	//arm state machine
	g_stateMachineArm1 : INT;
	g_stateMachineArm2 : INT;
	
	// index(0 to 4) of slave arm which is tele-linked to master arm
	g_teleSlaveArm1Idx : INT;
	g_teleSlaveArm2Idx : INT;
	
	//slave check enable  : true start , false end
	g_slaveCheckEnbale : BOOL;

	//0: init status 1: checking 2:check succeed 3: check failed
	g_slaveCheckStatus : UINT;

	//arm switch 
	g_armSwitchEnable : UINT:=0;

	//master hearbeat  : 1s frequency
	g_heartBeat : INT;

	//screen Lock Enable : true Lock  ,  false  unlock
	g_screenLockEnable : BOOL;
END_VAR

// ---- GVLs/GVL_MathDefine.TcGVL
VAR_GLOBAL CONSTANT
	g_smallNum :LREAL := 1E-8;
	g_smallAng :LREAL := 0.0001*PI/180;
	g_largeNum: LREAL :=1E16;
	g_deg2Rad :LREAL := pi/180.0;
	g_rad2Deg :LREAL := 180.0/pi;
	g_2pi :LREAL := 2*PI;
	
	g_eye3d :Mat3d:=[1, 0, 0,
					 0, 1, 0,
					 0, 0, 1];
	g_eye4d :Mat4d:=[1, 0, 0, 0,
					 0, 1, 0, 0,
					 0, 0, 1, 0,
					 0, 0, 0, 1];
	g_zeroMat3d :Mat3d:=[9(0)];
	
	g_zeroMat6d :Mat6d:=[36(0)];
	g_zeroMat7d :Mat7d:=[49(0)];
	g_eye7d :Mat7d:=[1, 0, 0, 0, 0, 0, 0, 
					 0, 1, 0, 0, 0, 0, 0, 
					 0, 0, 1, 0, 0, 0, 0, 
					 0, 0, 0, 1, 0, 0, 0,
					 0, 0, 0, 0, 1, 0, 0,
					 0, 0, 0, 0, 0, 1, 0,
					 0, 0, 0, 0, 0, 0, 1];
	
	g_zeroVec3d :Vec3d:= [3(0)];
	g_onesVec3d: Vec3d:=[3(1)];
	
	g_zeroVec6d: Vec6d:=[6(0)];
	g_onesVec6d: Vec6d:=[6(1)];
	
	g_zeroVec4d: Vec4d:=[4(0)];
	g_onesVec4d: Vec4d:=[4(1.0)];
	g_zeroVec4i: Vec4i:=[4(0)];
	g_onesVec4i: Vec4i:=[4(1)];
	
	g_zeroVec7d: Vec7d:=[7(0)];
	g_onesVec7d: Vec7d:=[7(1.0)];
	g_zeroVec7i: Vec7i:=[7(0)];
	g_onesVec7i: Vec7i:=[7(1)];
	
	g_allPosMode:Vec7i:=[7(DriverOPMode_Pos)];
	g_allTrqMode:Vec7i:=[7(DriverOPMode_Trq)];
	g_allPosTrqMode:Vec7i:=[7(DriverOPMode_PosTrq)];
	
	
END_VAR

// ---- GVLs/GVL_SafetyParameters.TcGVL
{attribute 'global_init_slot' := '49991'}
//TODO: safety check parameters need to be reviewd
VAR_GLOBAL CONSTANT
	
	// safety error counts threshold to trigger fault
	g_faultTriggerCounts :INT :=2;
	
	// arm joint safety error
	g_armMaxJntEncErr :vec7d:=[7(40*g_deg2Rad)];
	g_armMaxJntFollowErr :vec7d:=[7(20*g_deg2Rad)];
	
	// joint limit buffer(outside of joint limit)
	g_armJntPosLimitBuffer :vec7d:=[3(10.0*g_deg2Rad), 4(45.0*g_deg2Rad)];

	//max joint encoder current  saltation
	g_maxJntCurSalta : vec7di:=[7(60000)];
	
	// self check timeout time limit
	g_selfCheckTimeLimit : LREAL:= 15.0;
	
	//arm joint link encoder maximum and minimum values
	g_maxLinkEnc : DINT:=16777215;
	g_minLinkEnc : DINT:=0;
	
	//drive error word
	g_driveErrWord : UDINT:=32;
	
	// master arm cartesion control safety error 
	g_maxCartPosErr :LREAL := 0.005;
	g_maxCartOriErr :LREAL := 5.0*g_deg2Rad;
	

	// master joint safety error
	g_maxJntCtrlErr :LREAL := 15.0*g_deg2Rad;
	g_maxJntEncErr :LREAL := 30.0*g_deg2Rad;
	
	g_minJntPos: ARRAY[1..2,1..7] OF LREAL:=[-60*g_deg2Rad,	-45*g_deg2Rad-pi/2,		-45*g_deg2Rad, 	0, 	-135*g_deg2Rad+pi,		-45*g_deg2Rad-pi/2,		-g_largeNum,
											 -60*g_deg2Rad,	-45*g_deg2Rad-pi/2,		-45*g_deg2Rad,	0,		-135*g_deg2Rad+pi,		-45*g_deg2Rad+pi/2,	-g_largeNum];
	g_maxJntPos: ARRAY[1..2,1..7] OF LREAL:=[60*g_deg2Rad,	60*g_deg2Rad-pi/2,		60*g_deg2Rad,		2*pi,			135*g_deg2Rad+pi,		45*g_deg2Rad-pi/2,		g_largeNum,
								             60*g_deg2Rad,	60*g_deg2Rad-pi/2,		60*g_deg2Rad,		2*pi,			135*g_deg2Rad+pi,		45*g_deg2Rad+pi/2,		g_largeNum];

	
	// cart joint safety error
	g_cartMaxJntCtrlErr :Vec4d := [0.005, 5*g_deg2Rad,0.005, 0.005];
	g_cartMaxJntEncErr :Vec4d :=  [0.005, 5*g_deg2Rad,0.005, 0.005];

	// cart joint limit buffer(outside of joint limit)
	g_cartJntPosLimitBuffer :Vec4d :=[0.05, 10*g_deg2Rad,0.05, 0.05];
	
	// cart joint velocity limit
	g_cartMaxJntVel :Vec4d :=[0.03, 4*g_deg2Rad,0.02,0.015];
	
	// cart joint limit
	g_cartMinJntLimit : Vec4d :=[0-0.1, -(0+5)*g_deg2Rad, 0-0.1, 0-0.1];
	g_cartMaxJntLimit : Vec4d :=[0.38+0.1, (30+5)*g_deg2Rad, 0.24+0.1, 0.2+0.1];
	
	//cart joint follow error
	g_cartMaxJntFollowErr : Vec4d :=[0.01, 5*g_deg2rad, 0.01, 0.01];
	
	//cart joint current limit
	g_cartMaxJntCurrent : Vec4d :=[3800*2,3800*2,3800*2,3800*2];
	
	//cart joint encoder detetion value
	g_cartMaxLinkEnc : ARRAY [1..4] OF DINT := [67108863,16777215,67108863,67108863];
	g_cartMinLinkEnc : ARRAY [1..4] OF DINT := [4(0)];
END_VAR

VAR_GLOBAL
	//motor current limit
	g_motorCurrentLimit : Vec7d ;	

	g_arrayErrCodeArm:ARRAY [1..g_maxNum] OF ARRAY [0..100] OF UDINT;	
END_VAR

VAR_GLOBAL CONSTANT
	g_maxNum:INT:=3;
	g_maxArmNum:INT:=2;
	g_maxArmJoint:INT:=7; g_maxCartJoint:INT:=4;
	g_cartNum:UDINT:=3;
	MAX_CSV_ROWS 			: UDINT := 10000;(*最大行数(任务周期为20ms)即10分钟的buffer*)
	MAX_CSV_COLUMNS 		: UDINT := 130;(*最大列数*)
	MAX_CSV_FIELD_LENGTH	: UDINT := 35;(*每个字段的字符长度*)
	MAX_CSV_RING_BUFFER		: UDINT := 3;
	g_ArmNetID: ARRAY[1..g_maxArmNum] OF T_AmsNetId:=['192.168.0.10.4.1','192.168.0.10.9.1'];
	g_JointNetPort:ARRAY[1..g_maxArmNum,1..g_maxArmJoint] OF UINT :=[
											1001,    1002,	1003,	1004,	1005,	1006,	1007,
											1012,    1013,	1014,	1015,	1016,	1017,	1018	];
	g_cartNetID : T_AmsNetId := '192.168.0.10.9.1';
	g_cartJointNetPort:ARRAY[1..g_maxCartJoint] OF UINT :=[1008,    1009,	1010,	1011];
	
END_VAR

// ---- GVLs/GVL_SystemParameters.TcGVL
VAR_GLOBAL CONSTANT
	
	g_mArmNum :INT := 2;	
	g_mJntNum :INT := 7;	
	g_sArmNum :INT := 4;	
	g_sJntNum :INT := 11;
	g_cartDofs :INT :=6;
	
	
	
	// control loop interval for each task
	g_armCtrlCycleTime :LREAL :=0.00025;
	g_armCtrlFreq :LREAL :=1.0/g_armCtrlCycleTime;
	g_armDynamicCycleTime :LREAL := 0.001;
	g_armDynamicFreq :LREAL := 1.0/g_armDynamicCycleTime;
	g_cartCtrlCycleTime :LREAL := 0.001;
	g_cartCtrlFreq :LREAL := 1.0/g_cartCtrlCycleTime;
	
	// wait time before robot init  for ethercat to stablize 
	g_robotInitWaitTime : LREAL := 1.0;
	g_robotSafetyCheckWaitTime : LREAL :=3.0;
END_VAR

// ---- FBs_StateControllers/I_MasterArmCtrl.TcIO
INTERFACE I_MasterArmCtrl

METHOD init : BOOL
VAR_IN_OUT CONSTANT
	i_masterArm	:FB_MasterArm;
END_VAR
VAR_IN_OUT 
	r_masterArmCtrlCmd :ST_ArmCtrlCmds;
END_VAR
END_METHOD

PROPERTY isFinished : bool
GET
END_GET
END_PROPERTY

METHOD reset : BOOL
VAR_INPUT
END_VAR
END_METHOD

METHOD run : BOOL

VAR_IN_OUT CONSTANT
	i_slaveIdx :INT;
	i_shoulderPose :ST_Frame;
	i_masterArm :FB_MasterArm;
	i_slaveStatus :ST_SlaveStatus;
END_VAR
VAR_IN_OUT
	r_masterArmCtrlCmd :ST_ArmCtrlCmds;
END_VAR
END_METHOD

END_INTERFACE

// ---- Mains/MasterArmControl.TcPOU
PROGRAM MasterArmControl
VAR
	// slave robot data, input from slave controller box
	m_slaveRobotData AT %I* : MSCommu_slaveStatus;
	
	// all data from other tasks and controller 
	m_masterInputDataPool : ST_MasterInputDataPool;
	
	// master robot information, including arm status and cartesian data, output to other tasks
	m_masterStatus AT %Q* :ST_MasterStatus;
	
	// master robot joint data, output to other tasks
	m_masterJointsData AT %Q* :ST_MasterJointData;
		
	// master robot data, ouput to slave controller box
	m_masterRobotData AT %Q* :MSCommu_MasterStatus;
	
	// flag to init robot
	m_robotInit :BOOL :=FALSE;
	
	// wait time before robot init  for ethercat to be statble 
	m_robotInitWaitTime : LREAL:=0;
	
	// master robot
	m_masterRobot:FB_MasterRobot;
	
	// code execute time measure
	m_codeTime : Profiler;
	
END_VAR

m_codeTime(START:=TRUE, RESET:=TRUE);

// wait communication to be stable
IF(m_robotInitWaitTime<g_robotInitWaitTime) THEN
	m_robotInitWaitTime := m_robotInitWaitTime+g_armCtrlCycleTime;
	RETURN;
END_IF

// robot init
IF m_robotInit =FALSE THEN
	m_masterRobot.Init();
	m_robotInit:=TRUE;
END_IF

// input from UI
UIInputProcess();

// slave input data cast
slaveInputDataCast(m_slaveRobotData, m_masterInputDataPool.m_slaveStatus);

// robot run
m_masterRobot.run(m_masterInputDataPool);

// update data pool
m_masterRobot.getStatus(m_masterStatus,m_masterJointsData);

// master output data cast
masterOutputDataCast(m_masterRobot.m_shoulderPoseInMonitor, m_masterStatus, m_masterRobotData);

// output to UI
UIOutputProcess();

m_codeTime(START:=FALSE);

// convert from local ST_MasterStatus for control to MSCommu_MasterStatus for master-slave communication
METHOD masterOutputDataCast : BOOL
VAR_IN_OUT CONSTANT
	shoulderPose :ARRAY[1..2] OF ST_Frame;
	masterStatus :ST_MasterStatus;
END_VAR
VAR_IN_OUT
	masterOutputData:MSCommu_MasterStatus;
END_VAR

VAR
	i,j : INT;
	poseInMonitor:ST_Frame;
	velInShoulder, wVelInShoulder :Vec3d;
	velInMonitor, wVelInMonitor :Vec3d;
END_VAR
// Master heart beat
IF masterOutputData.m_heartBeat >= 10 THEN
	masterOutputData.m_heartBeat := 0;
ELSE
	masterOutputData.m_heartBeat := masterOutputData.m_heartBeat + 1;
END_IF

masterOutputData.m_motionScale :=masterStatus.m_motionScale;
masterOutputData.m_slaveSelfCheckFlag := m_masterInputDataPool.m_UIData.m_selfCheckFlag;
masterOutputData.m_pedalHover := m_masterInputDataPool.m_cartStatus.m_pedalHover;
masterOutputData.m_electricKnifePedalTrigger := m_masterInputDataPool.m_cartStatus.m_electricKnifePedalTrigger;
masterOutputData.m_tryMSControl[1] := BOOL_TO_INT(m_masterInputDataPool.m_cartStatus.m_surgonReady);
masterOutputData.m_tryMSControl[2] := BOOL_TO_INT(m_masterInputDataPool.m_cartStatus.m_surgonReady);
masterOutputData.m_uiResetFault := GVL_interactUI.g_uiResetFault;
masterOutputData.m_masterStopButton := NOT SafetyCheck.m_stopButton;

FOR i:=1 TO g_mArmNum DO
	masterOutputData.m_armState[i] := masterStatus.m_armState[i];
	masterOutputData.m_teleSlaveArmIdx[i] :=masterStatus.m_teleSlaveArmIdx[i];
	masterOutputData.m_gripAngle[i] := masterStatus.m_gripAngle[i] ;
	
	poseInMonitor := transform(shoulderPose[i],  masterStatus.m_curArmPose[i]);
	masterOutputData.m_curArmPose[i].m_pos := poseInMonitor.m_pos ;
	masterOutputData.m_curArmPose[i].m_rot := poseInMonitor.m_rot ;
	
	FOR j:=1 TO 3 DO
		velInShoulder[j]:=masterStatus.m_curArmTwist[i][j];
		wVelInShoulder[j]:=masterStatus.m_curArmTwist[i][j+3];
	END_FOR
	matMultiVec(shoulderPose[i].m_rot, velInShoulder,velInMonitor);
	matMultiVec(shoulderPose[i].m_rot, wVelInShoulder,wVelInMonitor);
	
	FOR j:=1 TO 3 DO
		masterOutputData.m_curArmTwist[i][j]:=velInMonitor[j];
		masterOutputData.m_curArmTwist[i][j+3]:=wVelInMonitor[j];
	END_FOR
END_FOR
END_METHOD

// convert from MSCommu_Slavetatus for master-slave communication to local ST_SlaveStatus for control
METHOD slaveInputDataCast : BOOL
VAR_IN_OUT CONSTANT
		slaveInputData : MSCommu_SlaveStatus; 
END_VAR
VAR_IN_OUT
	slaveStatus :ST_SlaveStatus;
END_VAR

VAR
	i :INT;
END_VAR
slaveStatus.m_selfCheckPass := slaveInputData.m_selfCheckPass;
slaveStatus.m_slaveHeartBeat := slaveInputData.m_heartBeat;
slaveStatus.m_endoscopeMounted :=slaveInputData.m_endoscopeMounted;
slaveStatus.m_endoscopePose.m_pos :=slaveInputData.m_endoscopePose.m_pos;
slaveStatus.m_endoscopePose.m_rot :=slaveInputData.m_endoscopePose.m_rot;
slaveStatus.m_asepticDeployCompleteFlag := slaveInputData.m_asepticDeployCompletedFlag;
slaveStatus.m_slaveStopButton := slaveInputData.m_slaveStopButton;
FOR i:= 1 TO g_sArmNum DO
	slaveStatus.m_armState[i] := slaveInputData.m_armState[i];
	slaveStatus.m_instruStauts[i].m_fingerAngle := slaveInputData.m_instruStauts[i].m_fingerAngle;
	slaveStatus.m_instruStauts[i].m_ready := slaveInputData.m_instruStauts[i].m_ready;
	slaveStatus.m_instruStauts[i].m_type := slaveInputData.m_instruStauts[i].m_type;
	slaveStatus.m_instruStauts[i].m_energyType := slaveInputData.m_instruEnergyType[i];
	slaveStatus.m_curArmPose[i].m_pos :=slaveInputData.m_curArmPose[i].m_pos;
	slaveStatus.m_curArmPose[i].m_rot :=slaveInputData.m_curArmPose[i].m_rot;
	slaveStatus.m_masterSlavePoseError[i] := slaveInputData.m_masterSlavePoseError[i];
END_FOR
END_METHOD

// tranform data from UI(global variable write by ADS) to ST_UIData
METHOD UIInputProcess : BOOL
VAR_INPUT
END_VAR
// master-slave control scale
IF 2 = GVL_interactUI.g_masterSlaveScaling THEN
	m_masterInputDataPool.m_UIData.m_motionScale := 2;
ELSIF 3 = GVL_interactUI.g_masterSlaveScaling THEN
	m_masterInputDataPool.m_UIData.m_motionScale := 3;
ELSE
	m_masterInputDataPool.m_UIData.m_motionScale := 1.5;
END_IF

// self-check
m_masterInputDataPool.m_UIData.m_selfCheckFlag := GVL_interactUI.g_slaveCheckEnbale;

// hand clutch
m_masterInputDataPool.m_UIData.m_enableHandClutch := GVL_interactUI.g_fingerClutchOnOff;

// arm disable
m_masterInputDataPool.m_UIData.m_masterArmDisableFlag[1]:=FALSE;
m_masterInputDataPool.m_UIData.m_masterArmDisableFlag[2]:=FALSE;
IF 1=GVL_interactUI.g_armIsDisbale OR 2=GVL_interactUI.g_armIsDisbale THEN
	m_masterInputDataPool.m_UIData.m_masterArmDisableFlag[GVL_interactUI.g_armIsDisbale] := TRUE;
END_IF
END_METHOD

METHOD UIOutputProcess : BOOL
VAR_INPUT
END_VAR
//TODO
//slave arm self check status
IF m_masterInputDataPool.m_slaveStatus.m_armState[1] = SlaveArmState_SelfCheck OR m_masterInputDataPool.m_slaveStatus.m_armState[2] = SlaveArmState_SelfCheck OR 
			m_masterInputDataPool.m_slaveStatus.m_armState[3] = SlaveArmState_SelfCheck OR m_masterInputDataPool.m_slaveStatus.m_armState[4] = SlaveArmState_SelfCheck THEN
	GVL_interactUI.g_slaveCheckStatus := 1;
ELSIF m_masterInputDataPool.m_slaveStatus.m_selfCheckPass THEN
	GVL_interactUI.g_slaveCheckStatus := 2;
ELSE
	GVL_interactUI.g_slaveCheckStatus := 0;
END_IF

//GVL_interactUI.g_masterSelfCheckFinshed := m_masterStatus.m_selfCheckStatus;

GVL_interactUI.g_stateMachineArm1 := m_masterStatus.m_armState[1];
GVL_interactUI.g_stateMachineArm2 := m_masterStatus.m_armState[2];
GVL_interactUI.g_teleSlaveArm1Idx := m_masterStatus.m_teleSlaveArmIdx[1];
GVL_interactUI.g_teleSlaveArm2Idx := m_masterStatus.m_teleSlaveArmIdx[2];
GVL_interactUI.g_screenLockEnable := (MasterArmState_MasterSlave <= m_masterStatus.m_armState[1]  AND MasterArmState_Endoscope >= m_masterStatus.m_armState[1]) OR (MasterArmState_MasterSlave <= m_masterStatus.m_armState[2]  AND MasterArmState_Endoscope >= m_masterStatus.m_armState[2]);
IF m_masterInputDataPool.m_cartStatus.m_armSwitch THEN
	// ui reset variable
	GVL_interactUI.g_armSwitchEnable := 1;
END_IF

GVL_interactUI.g_plcVersion := '1(1.0.0.1)';
END_METHOD

END_PROGRAM

// ---- FBs_Robots/FB_MasterRobot.TcPOU
FUNCTION_BLOCK FB_MasterRobot
VAR
	// flag if slave are connected
	m_slaveOnLine :BOOL :=FALSE;
	m_slaveOnLineCheck :FB_slaveConnectionCheck;
	
	// master-slave motion scale
	m_motionScale :LREAL;
	
	// monitor angle
	m_monitorAngle :LREAL;
	
	// master arm base pose(shoulder pose) in monitor coordinate
	m_shoulderPoseInMonitor :ARRAY[1..2] OF ST_Frame;
	
	// master arms, responsible for arm kinematic and control
	m_masterArms :ARRAY[1..g_mArmNum] OF FB_MasterArm;
	
	// arm state
	m_masterArmState:ARRAY[1..g_mArmNum] OF E_masterArmState:=[E_masterArmState.MasterArmState_Init,E_masterArmState.MasterArmState_Error];
	m_lastMasterArmState:ARRAY[1..g_mArmNum] OF E_masterArmState:=[E_masterArmState.MasterArmState_Init,E_masterArmState.MasterArmState_Error];
	m_nextMasterArmState:ARRAY[1..g_mArmNum] OF E_masterArmState:=[E_masterArmState.MasterArmState_Init,E_masterArmState.MasterArmState_Error];
	
	// index(1 to 4) of slave arm which is tele-linked to master arm
	m_teleSlaveArmIdx:ARRAY[1..g_mArmNum] OF E_MatchedSlaveArmIdx:=[MatchedSlaveArmIdx_NULL, MatchedSlaveArmIdx_null];
	m_matchedMasterArmIdx :ST_MatchedMasterArmIdx;
	m_instruArmState:ARRAY [1..g_mArmNum] OF E_SlaveArmState:=[SlaveArmState_Error, SlaveArmState_Error];
	m_scopeArmState :E_SlaveArmState := SlaveArmState_Error;
	m_scopeArmIndex : E_MatchedSlaveArmIdx :=MatchedSlaveArmIdx_null;
	
	// flag if tele-manipulated slave arm is switched
	m_armSwitchFlag :ARRAY[1..2] OF BOOL := [2(FALSE)];
	
	// flag to enter master-slave control, triggerd by pinching the gripper twice in on second
	m_MSCtrlTriggerFlag :ARRAY[1..g_mArmNum] OF BOOL:=[FALSE, FALSE];
	m_MSCtrlTriggerCheck :ARRAY[1..g_mArmNum] OF FB_MSCtrlTriggerCheck;
	
	// all arm controller instance 
	m_armCtrlFactory :ARRAY[1..g_mArmNum,1..MasterArmState_totalNum] OF I_MasterArmCtrl;
	m_armError :ARRAY[1..g_mArmNum] OF FB_StateCtrlError;
	m_armInit :ARRAY[1..g_mArmNum] OF FB_StateCtrlInit;
	m_armHome :ARRAY[1..g_mArmNum] OF FB_StateCtrlHome;
	m_armStandBy :ARRAY[1..g_mArmNum] OF FB_StateCtrlStandBy;
	m_armMatching :ARRAY[1..g_mArmNum] OF FB_StateCtrlMatching;
	m_armReady :ARRAY[1..g_mArmNum] OF FB_StateCtrlReady;
	m_armMasterSlave :ARRAY[1..g_mArmNum] OF FB_StateCtrlMasterSlave;
	m_armClutch :ARRAY[1..g_mArmNum] OF FB_StateCtrlClutch;
	m_armEndoscope :ARRAY[1..g_mArmNum] OF FB_StateCtrlEndoscope;
	m_armCart :ARRAY[1..g_mArmNum] OF FB_StateCtrlCart;
	m_armGravityCali :ARRAY[1..g_mArmNum] OF FB_StateCtrlGraCali;
	m_armTest :ARRAY[1..g_mArmNum] OF FB_StateCtrlTest;
	m_armDisable :ARRAY[1..g_mArmNum] OF FB_StateCtrlDisable;
	m_armPerformance :ARRAY[1..g_mArmNum] OF FB_StateCtrlPerformance;
	
	// specialized endoscope controller
	m_scopeCtrl :FB_EndoscopeController;
	
	// arm controller interface
	m_armCtrl :ARRAY[1..g_mArmNum] OF I_MasterArmCtrl;
	m_armCtrlCmds :ARRAY[1..g_mArmNum] OF ST_ArmCtrlCmds;
	
	// ultrasonic knife rotation clutch flag
	m_USKnifeRotClutch :ARRAY[1..g_sArmNum] OF BOOL := [4(FALSE)];

END_VAR

 METHOD PROTECTED checkTeleSlaveArmIdx : BOOL
VAR_IN_OUT CONSTANT
	i_masterInputDataPool:ST_MasterInputDataPool;
END_VAR
VAR_STAT
	m_armSwitchR : R_TRIG;
	m_armSwitch : BOOL;
	nextTeleSlaveArmIdx:ARRAY[1..g_mArmNum] OF E_MatchedSlaveArmIdx;
END_VAR
nextTeleSlaveArmIdx:=m_teleSlaveArmIdx;
m_armSwitchR(CLK:= i_masterInputDataPool.m_cartStatus.m_armSwitch, Q=> m_armSwitch);
IF m_armSwitch THEN
	m_matchedMasterArmIdx.left1ArmIdx := GVL_interactUI.g_armDistributionInfo.m_leftMappingSlaveArm[1];
	m_matchedMasterArmIdx.left2ArmIdx := GVL_interactUI.g_armDistributionInfo.m_leftMappingSlaveArm[2];
	m_matchedMasterArmIdx.right1ArmIdx := GVL_interactUI.g_armDistributionInfo.m_rightMappingSlaveArm[1];
	m_matchedMasterArmIdx.right2ArmIdx := GVL_interactUI.g_armDistributionInfo.m_rightMappingSlaveArm[2];
END_IF


IF m_matchedMasterArmIdx.left1ArmIdx <=0 OR m_matchedMasterArmIdx.left2ArmIdx <=0 OR m_matchedMasterArmIdx.right1ArmIdx <=0 OR m_matchedMasterArmIdx.right2ArmIdx <=0 THEN
	RETURN;
END_IF

// switch tele-controlled arm index when arm is disenabled
IF i_masterInputDataPool.m_slaveStatus.m_armState[m_matchedMasterArmIdx.left1ArmIdx] = SlaveArmState_Disable THEN
	nextTeleSlaveArmIdx[1]:= m_matchedMasterArmIdx.left2ArmIdx;
ELSIF i_masterInputDataPool.m_slaveStatus.m_armState[m_matchedMasterArmIdx.left2ArmIdx] = SlaveArmState_Disable THEN
	nextTeleSlaveArmIdx[1]:= m_matchedMasterArmIdx.left1ArmIdx;
ELSIF i_masterInputDataPool.m_slaveStatus.m_armState[m_matchedMasterArmIdx.right1ArmIdx] = SlaveArmState_Disable THEN
	nextTeleSlaveArmIdx[2]:= m_matchedMasterArmIdx.right2ArmIdx;
ELSIF i_masterInputDataPool.m_slaveStatus.m_armState[m_matchedMasterArmIdx.right2ArmIdx] = SlaveArmState_Disable THEN
	nextTeleSlaveArmIdx[2]:= m_matchedMasterArmIdx.right1ArmIdx;
END_IF


// switch tele-controlled arm index when endoscope is mounted
IF m_scopeArmIndex = m_matchedMasterArmIdx.left1ArmIdx OR m_scopeArmIndex = m_matchedMasterArmIdx.left2ArmIdx THEN
	// left arm
	IF m_scopeArmIndex = m_matchedMasterArmIdx.left1ArmIdx THEN
		nextTeleSlaveArmIdx[1] := m_matchedMasterArmIdx.left2ArmIdx;
	ELSE
		nextTeleSlaveArmIdx[1] := m_matchedMasterArmIdx.left1ArmIdx;
	END_IF
	
	// right arm
	// switch tele-controlled arm index when arm switch is triggerd
	IF m_armSwitch THEN
		IF m_teleSlaveArmIdx[2] = m_matchedMasterArmIdx.right1ArmIdx AND i_masterInputDataPool.m_slaveStatus.m_armState[m_matchedMasterArmIdx.right2ArmIdx]=SlaveArmState_InstruReady THEN
			nextTeleSlaveArmIdx[2] := m_matchedMasterArmIdx.right2ArmIdx;
		ELSIF 
			m_teleSlaveArmIdx[2]=m_matchedMasterArmIdx.right2ArmIdx AND i_masterInputDataPool.m_slaveStatus.m_armState[m_matchedMasterArmIdx.right1ArmIdx]=SlaveArmState_InstruReady THEN
			nextTeleSlaveArmIdx[2] := m_matchedMasterArmIdx.right1ArmIdx;
		ELSE
			IF  i_masterInputDataPool.m_slaveStatus.m_armState[m_matchedMasterArmIdx.right1ArmIdx]=SlaveArmState_InstruReady THEN
				nextTeleSlaveArmIdx[2] := m_matchedMasterArmIdx.right1ArmIdx;
			ELSIF i_masterInputDataPool.m_slaveStatus.m_armState[m_matchedMasterArmIdx.right2ArmIdx]=SlaveArmState_InstruReady THEN
				nextTeleSlaveArmIdx[2] := m_matchedMasterArmIdx.right2ArmIdx;
			ELSE
				nextTeleSlaveArmIdx[2] := m_matchedMasterArmIdx.right1ArmIdx;
			END_IF
			
		END_IF
	END_IF

ELSIF m_scopeArmIndex = m_matchedMasterArmIdx.right1ArmIdx OR m_scopeArmIndex = m_matchedMasterArmIdx.right2ArmIdx THEN
	// left arm
	// switch tele-controlled arm index when arm switch is triggerd
	IF m_armSwitch THEN
		IF m_teleSlaveArmIdx[1]=m_matchedMasterArmIdx.left1ArmIdx AND i_masterInputDataPool.m_slaveStatus.m_armState[m_matchedMasterArmIdx.left2ArmIdx]=SlaveArmState_InstruReady THEN
			nextTeleSlaveArmIdx[1] := m_matchedMasterArmIdx.left2ArmIdx;
		ELSIF 
			m_teleSlaveArmIdx[1]=m_matchedMasterArmIdx.left2ArmIdx AND i_masterInputDataPool.m_slaveStatus.m_armState[m_matchedMasterArmIdx.left1ArmIdx]=SlaveArmState_InstruReady THEN
			nextTeleSlaveArmIdx[1] := m_matchedMasterArmIdx.left1ArmIdx;
		ELSE
			IF  i_masterInputDataPool.m_slaveStatus.m_armState[m_matchedMasterArmIdx.left1ArmIdx]=SlaveArmState_InstruReady THEN
				nextTeleSlaveArmIdx[1] := m_matchedMasterArmIdx.left1ArmIdx;
			ELSIF i_masterInputDataPool.m_slaveStatus.m_armState[m_matchedMasterArmIdx.left2ArmIdx]=SlaveArmState_InstruReady THEN
				nextTeleSlaveArmIdx[1] := m_matchedMasterArmIdx.left2ArmIdx;
			ELSE
				nextTeleSlaveArmIdx[1] := m_matchedMasterArmIdx.left1ArmIdx;
			END_IF
		END_IF
	END_IF

	// right arm
	IF m_scopeArmIndex = m_matchedMasterArmIdx.right1ArmIdx THEN
		nextTeleSlaveArmIdx[2] := m_matchedMasterArmIdx.right2ArmIdx;
	ELSE
		nextTeleSlaveArmIdx[2] := m_matchedMasterArmIdx.right1ArmIdx;
	END_IF
END_IF

// check if arm-switch is triggerd
m_armSwitchFlag[1]:=m_teleSlaveArmIdx[1] <>  nextTeleSlaveArmIdx[1];
m_armSwitchFlag[2]:=m_teleSlaveArmIdx[2] <>  nextTeleSlaveArmIdx[2];

m_teleSlaveArmIdx:= nextTeleSlaveArmIdx;
END_METHOD

METHOD PROTECTED controllerTransit : BOOL
VAR_INPUT
END_VAR
VAR
	i :INT;
END_VAR
FOR i:=1 TO g_mArmNum DO 
	IF m_nextMasterArmState[i]<> m_masterArmState[i] THEN
		// reset current controller
		m_armCtrl[i].reset();
		
		// transit to new controller
		m_lastMasterArmState[i]:=m_masterArmState[i];
		m_masterArmState[i]:=m_nextMasterArmState[i];
		m_armCtrl[i]:=m_armCtrlFactory[i,m_masterArmState[i]];
		
		// init next controller
		m_armCtrl[i].Init(m_masterArms[i],m_armCtrlCmds[i]);
		
		// init scope controller
		IF m_masterArmState[i] = MasterArmState_Endoscope  THEN
			m_scopeCtrl.init(m_shoulderPoseInMonitor, m_masterArms, m_armCtrlCmds);
		END_IF
		
		m_masterArms[i].updateCmds(m_armCtrlCmds[i]);
	END_IF
END_FOR
END_METHOD

METHOD PUBLIC getStatus : BOOL
VAR_IN_OUT
	// master robot information, including arm status and cartesian data
	r_masterStatus :ST_MasterStatus;
	
	// master robot joint data
	r_masterJointsData :ST_MasterJointData;
	
END_VAR

VAR
	i:INT;
END_VAR
r_masterStatus.m_motionScale := m_motionScale;
r_masterStatus.m_armState:=m_masterArmState;
r_masterStatus.m_teleSlaveArmIdx := m_teleSlaveArmIdx;
r_masterStatus.m_matchedMasterArmIdx := m_matchedMasterArmIdx;

FOR i:=1 TO g_mArmNum DO
	// current info
	r_masterStatus.m_gripAngle[i]:=m_masterArms[i].gripAngle;
	// cartesion
	r_masterStatus.m_curArmPose[i]:=m_masterArms[i].curCartPose;
	r_masterStatus.m_curArmTwist[i]:=m_masterArms[i].curCartTwist;
	// joint
	r_masterJointsData.m_curMotorPos[i]:=m_masterArms[i].curMotorPos;
	r_masterJointsData.m_curLinkPos[i]:=m_masterArms[i].curLinkPos;
	r_masterJointsData.m_curJntPos[i]:=m_masterArms[i].curJntPos;
	r_masterJointsData.m_curJntVel[i]:=m_masterArms[i].curJntVel;
	r_masterJointsData.m_curJntTrq[i]:=m_masterArms[i].curJntTrq;
	r_masterJointsData.m_rawJntCurrent[i]:=m_masterArms[i].rawJntCurrent;
	r_masterJointsData.m_filtJntCurrent[i]:=m_masterArms[i].filtJntCurrent;
	
	// command info
	// cartesion
	r_masterStatus.m_cmdArmPose[i]:=m_masterArms[i].m_cmdCartPose;
	r_masterStatus.m_cmdArmTwist[i]:=m_masterArms[i].m_cmdCartTwist;
	// joint info
	r_masterJointsData.m_cmdJntPos[i]:=m_masterArms[i].m_cmdJntPos;
	r_masterJointsData.m_cmdJntVel[i]:=m_masterArms[i].m_cmdJntVel;
	r_masterJointsData.m_cmdJntTrq[i]:=m_masterArms[i].m_cmdJntTrq;
	r_masterJointsData.m_cmdJntCurrent[i]:=m_masterArms[i].cmdJntCurrent;
	//data to safety check
	r_masterStatus.m_gripHallSensor[i] := m_masterArms[i].m_gripHallSensorIO;
	r_masterStatus.m_slaveOnLine := m_slaveOnLine;
	r_masterStatus.m_IKSuccess[i] := m_armMatching[i].IKSuccess;
	r_masterStatus.m_timePeriod[i] := m_armMatching[i].timePeriod;
	//r_masterStatus.m_selfCheckStatus
END_FOR
END_METHOD

METHOD PUBLIC Init : BOOL
VAR_INPUT
END_VAR
VAR
	i:INT;
END_VAR
// init tele-controlled arm index
m_teleSlaveArmIdx[1]:=MatchedSlaveArmIdx_1;
m_teleSlaveArmIdx[2]:=MatchedSlaveArmIdx_3;

// shoulder pose in monitor
m_shoulderPoseInMonitor[1].m_pos[1]:=-g_shoulderDistance/2;
m_shoulderPoseInMonitor[2].m_pos[1]:=g_shoulderDistance/2;

FOR i:=1 TO g_mArmNum DO
	// arm init
	m_masterArms[i].Init(i);
	m_masterArmState[i]:=MasterArmState_Init;
	m_lastMasterArmState[i]:=MasterArmState_Init;
	m_nextMasterArmState[i]:=MasterArmState_Init;
	
	// command init
	m_armCtrlCmds[i].m_jntEnableFlag := g_zeroVec7i;
	m_armCtrlCmds[i].m_jntOPMode := g_allPosMode;
	m_armCtrlCmds[i].m_cmdCartPose := m_masterArms[i].curCartPose;
	m_armCtrlCmds[i].m_cmdCartTwist := g_zeroVec6d;
	m_armCtrlCmds[i].m_cmdJntPos := m_masterArms[i].curJntPos;
	m_armCtrlCmds[i].m_cmdJntVel := g_zeroVec7d;
	m_armCtrlCmds[i].m_cmdJntAcc := g_zeroVec7d;
	m_armCtrlCmds[i].m_cmdJntTrq := g_zeroVec7d;
	
	// generate controller factory
	m_armCtrlFactory[i,MasterArmState_Error] := m_armError[i];
	m_armCtrlFactory[i,MasterArmState_Init] := m_armInit[i];
	m_armCtrlFactory[i,MasterArmState_Home] := m_armHome[i];
	m_armCtrlFactory[i,MasterArmState_Standby] := m_armStandBy[i];
	m_armCtrlFactory[i,MasterArmState_Matching] := m_armMatching[i];
	m_armCtrlFactory[i,MasterArmState_Ready] := m_armReady[i];
	m_armCtrlFactory[i,MasterArmState_MasterSlave] := m_armMasterSlave[i];
	m_armCtrlFactory[i,MasterArmState_Clutch] := m_armClutch[i];
	m_armCtrlFactory[i,MasterArmState_Endoscope] := m_armEndoscope[i];
	m_armCtrlFactory[i,MasterArmState_Cart] := m_armCart[i];
	m_armCtrlFactory[i,MasterArmState_GravityCali] := m_armGravityCali[i];
	m_armCtrlFactory[i,MasterArmState_Test] := m_armTest[i];
	m_armCtrlFactory[i,MasterArmState_Disable] := m_armDisable[i];
	m_armCtrlFactory[i,MasterArmState_Performance] := m_armPerformance[i];

	// assign controller
	m_armCtrl[i]:=m_armCtrlFactory[i,m_masterArmState[i]];
	m_armCtrl[i].Init(m_masterArms[i],m_armCtrlCmds[i]);
	
	// init master-slave trigger
	m_MSCtrlTriggerCheck[i].init(g_armCtrlCycleTime, 2);
END_FOR
END_METHOD

METHOD PROTECTED MSCtrlTriggerCheck : BOOL
VAR_IN_OUT CONSTANT
		i_masterInputDataPool:ST_MasterInputDataPool;
END_VAR
VAR
	i:INT;
END_VAR
FOR i:=1 TO g_mArmNum DO
	IF MasterArmState_Ready = m_masterArmState[i] AND SlaveArmState_InstruReady = m_instruArmState[i] 
		AND SlaveArmState_ScopeReady = m_scopeArmState AND i_masterInputDataPool.m_cartStatus.m_surgonReady THEN
		m_MSCtrlTriggerFlag[i]:=m_MSCtrlTriggerCheck[i].run(m_masterArms[i].gripAngle);
	END_IF
	
	IF  MatchedSlaveArmIdx_NULL =  m_teleSlaveArmIdx[i] OR   NOT(i_masterInputDataPool.m_cartStatus.m_surgonReady) 
		OR 	NOT(i_masterInputDataPool.m_slaveStatus.m_instruStauts[m_teleSlaveArmIdx[i]].m_ready) 
		OR m_masterArmState[i] = MasterArmState_Error
		OR  SlaveArmState_Error = m_instruArmState[i] OR SlaveArmState_Disable = m_instruArmState[i]  THEN
		m_MSCtrlTriggerFlag[i]:=FALSE;
		m_MSCtrlTriggerCheck[i].reset();
	END_IF  
END_FOR
END_METHOD

METHOD PUBLIC run : BOOL
VAR_IN_OUT CONSTANT
	i_masterInputDataPool:ST_MasterInputDataPool;
END_VAR
VAR
	i:INT;
END_VAR
m_motionScale := i_masterInputDataPool.m_UIData.m_motionScale;
m_monitorAngle := i_masterInputDataPool.m_cartStatus.m_monitorAngle;

// check slave connection
m_slaveOnLine := m_slaveOnLineCheck.check(i_masterInputDataPool.m_slaveStatus.m_slaveHeartBeat);

// update shoulder pose
updateShoulderPose();

// check tele-operated slave arms index
checkTeleSlaveArmIdx(i_masterInputDataPool);

// check if to trig ultrasonic knife ratotation clutch
USKnifeClutchCheck(i_masterInputDataPool);

// update arm status
FOR i:=1 TO g_mArmNum DO
	// update dynamic data
	m_masterArms[i].updateDyna(i_masterInputDataPool.m_masterDynaData);
								
	// update master arm kinematics
	m_masterArms[i].updateStatus();
END_FOR

// state machine transition
stateMachine(i_masterInputDataPool);

// controller transition
controllerTransit();

// run arm controller
FOR i:=1 TO g_mArmNum DO
	// null ptr check
	ASSERT(0 <> m_armCtrl[i]);
	
	// run controller
	m_armCtrl[i].run(m_teleSlaveArmIdx[i], m_shoulderPoseInMonitor[i], m_masterArms[i],
						i_masterInputDataPool.m_slaveStatus,m_armCtrlCmds[i]);
						
	// update commands to drivers
	m_masterArms[i].updateCmds(m_armCtrlCmds[i]);
END_FOR

// run scope controller
IF m_masterArmState[1] = MasterArmState_Endoscope AND m_masterArmState[2] = MasterArmState_Endoscope THEN
	m_scopeCtrl.run(m_teleSlaveArmIdx, m_shoulderPoseInMonitor, m_masterArms, i_masterInputDataPool.m_slaveStatus, m_armCtrlCmds);
	m_masterArms[1].updateCmds(m_armCtrlCmds[1]);
	m_masterArms[2].updateCmds(m_armCtrlCmds[2]);
END_IF
END_METHOD

PROPERTY shoulderPose : ARRAY[1..2] OF ST_Frame
GET
shoulderPose := m_shoulderPoseInMonitor;
END_GET
END_PROPERTY

// state machine check and transit 
METHOD PROTECTED stateMachine : BOOL
VAR_IN_OUT CONSTANT
		i_masterInputDataPool:ST_MasterInputDataPool;
END_VAR
VAR
	i:INT;
	enableClutch :BOOL;
END_VAR
// get instrument arm state
FOR i:=1 TO g_mArmNum DO
	IF MatchedSlaveArmIdx_NULL =  m_teleSlaveArmIdx[i] THEN
		m_instruArmState[i] := SlaveArmState_Error;
	ELSE
		m_instruArmState[i] := i_masterInputDataPool.m_slaveStatus.m_armState[m_teleSlaveArmIdx[i]];
	END_IF
END_FOR

// get endoscope arm state
m_scopeArmState := SlaveArmState_Error;
m_scopeArmIndex := MatchedSlaveArmIdx_null;
FOR i:=1 TO g_sArmNum DO 
	IF InstruType_endoscope =  i_masterInputDataPool.m_slaveStatus.m_instruStauts[i].m_type THEN
		m_scopeArmState := i_masterInputDataPool.m_slaveStatus.m_armState[i];
		m_scopeArmIndex := i;
		EXIT;
	END_IF
END_FOR

// check if master-slave grip angle match
MSCtrlTriggerCheck(i_masterInputDataPool);

// State machine transit 
FOR i:=1 TO g_mArmNum DO
	
	// flag if enable clutch
	enableClutch :=  i_masterInputDataPool.m_cartStatus.m_clutchSwitch OR (m_masterArms[i].handClutchSwitch AND i_masterInputDataPool.m_UIData.m_enableHandClutch);
	
	CASE m_masterArmState[i] OF
		// error
		MasterArmState_Error:
			// to standby
			IF FALSE = i_masterInputDataPool.m_safetyData.m_masterErrFlag[i] THEN
				m_nextMasterArmState[i] := MasterArmState_Standby;
			END_IF
			
		// init
		MasterArmState_Init:
			// to home
			IF m_armCtrl[i].isFinished THEN
				// NOTICE: multiple cycles joints back to center during initialization
				// 			need to reset joints encoder data again
				m_masterArms[i].initJntPos();
				m_nextMasterArmState[i]:=MasterArmState_Home;
			END_IF

		//home
		MasterArmState_Home:
			IF m_armCtrl[i].isFinished  THEN
				m_nextMasterArmState[i]:=MasterArmState_Standby;
			END_IF
		
		//standby
		MasterArmState_Standby:
			// to matching
			IF SlaveArmState_InstruReady = m_instruArmState[i] AND SlaveArmState_ScopeReady = m_scopeArmState THEN
				m_nextMasterArmState[i]:=MasterArmState_Matching;
			// to clutch
			ELSIF enableClutch THEN
				m_nextMasterArmState[i] := MasterArmState_Clutch; 
			// to cart
			ELSIF i_masterInputDataPool.m_cartStatus.m_consoleInAdjust THEN
				m_nextMasterArmState[i] := MasterArmState_Cart;
			END_IF
		
		//matching
		MasterArmState_Matching:
			// to ready
			IF m_armCtrl[i].isFinished THEN
				m_nextMasterArmState[i]:=MasterArmState_Ready;
			// to clutch
			ELSIF enableClutch THEN
				m_nextMasterArmState[i] := MasterArmState_Clutch; 
			// to standby
			ELSIF SlaveArmState_InstruReady <> m_instruArmState[i] OR SlaveArmState_ScopeReady <> m_scopeArmState
						OR m_armSwitchFlag[i] THEN
				m_nextMasterArmState[i]:=MasterArmState_Standby;
			// to cart
			ELSIF i_masterInputDataPool.m_cartStatus.m_consoleInAdjust THEN
				m_nextMasterArmState[i] := MasterArmState_Cart;
			END_IF
		
		//ready
		MasterArmState_Ready:
			// to standby
			IF SlaveArmState_InstruReady <> m_instruArmState[i] OR SlaveArmState_ScopeReady <> m_scopeArmState
					OR m_armSwitchFlag[i] THEN
				m_nextMasterArmState[i]:=MasterArmState_Standby;
			// to clutch
			ELSIF enableClutch THEN
				m_nextMasterArmState[i] := MasterArmState_Clutch; 
			// to cart
			ELSIF i_masterInputDataPool.m_cartStatus.m_consoleInAdjust THEN
				m_nextMasterArmState[i] := MasterArmState_Cart;
			// to master-slave
			ELSIF SlaveArmState_InstruReady = m_instruArmState[i] AND SlaveArmState_ScopeReady = m_scopeArmState 
					AND i_masterInputDataPool.m_cartStatus.m_surgonReady AND m_MSCtrlTriggerFlag[i] AND i_masterInputDataPool.m_slaveStatus.m_asepticDeployCompleteFlag THEN
				m_nextMasterArmState[i] := MasterArmState_MasterSlave;
			END_IF
		
		//MasterSlave
		MasterArmState_MasterSlave:
			// to standdy
			IF  (SlaveArmState_InstruReady <> m_instruArmState[i] AND SlaveArmState_MasterSlave <> m_instruArmState[i])
				OR SlaveArmState_ScopeReady <> m_scopeArmState OR NOT(i_masterInputDataPool.m_cartStatus.m_surgonReady)
				OR m_armSwitchFlag[i] THEN
				m_nextMasterArmState[i]:=MasterArmState_Standby;
			// to clutch
			ELSIF enableClutch THEN
				m_nextMasterArmState[i] := MasterArmState_Clutch; 
			END_IF
			
		//Clutch
		MasterArmState_Clutch:
			// to standby
			IF NOT(enableClutch) THEN
				m_nextMasterArmState[i]:=MasterArmState_Standby;
			END_IF
		
		// Endoscope 
		MasterArmState_Endoscope:
			// to standby
			IF NOT(i_masterInputDataPool.m_cartStatus.m_surgonReady) OR NOT(i_masterInputDataPool.m_cartStatus.m_endoscopeSwitch) 
				OR (SlaveArmState_ScopeReady <> m_scopeArmState AND SlaveArmState_EndoScope <> m_scopeArmState) THEN
				m_nextMasterArmState[i] := MasterArmState_Standby;
			// to clutch
			ELSIF enableClutch THEN
				m_nextMasterArmState[i] := MasterArmState_Clutch; 
			// to cart
			ELSIF i_masterInputDataPool.m_cartStatus.m_consoleInAdjust THEN
				m_nextMasterArmState[i] := MasterArmState_Cart;
			END_IF
			
		// Cart 
		MasterArmState_Cart:
			// to standby
			IF NOT( i_masterInputDataPool.m_cartStatus.m_consoleInAdjust) THEN
				m_nextMasterArmState[i] := MasterArmState_Standby;
			END_IF
		
		//Gravity Calibration
		MasterArmState_GravityCali:
			// to standby
			IF  m_armCtrl[i].isFinished THEN
				m_nextMasterArmState[i]:=MasterArmState_Standby;
			END_IF
	
		//arm test
		MasterArmState_Test:
			// to standby
			IF  m_armCtrl[i].isFinished THEN
				m_nextMasterArmState[i]:=MasterArmState_Standby;
			END_IF
			
		//arm Performance
		MasterArmState_Performance:
			// to standby
			IF  m_armCtrl[i].isFinished THEN
				m_nextMasterArmState[i]:=MasterArmState_Standby;
			END_IF
			
		//arm disable
		MasterArmState_Disable:
			// to init
			IF  NOT(i_masterInputDataPool.m_UIData.m_masterArmDisableFlag[i]) THEN
				m_nextMasterArmState[i]:=MasterArmState_Init;
			END_IF
	END_CASE
	
	// arm disable
	IF i_masterInputDataPool.m_UIData.m_masterArmDisableFlag[i] THEN
		m_nextMasterArmState[i] := MasterArmState_Disable;
	// error check
	ELSIF i_masterInputDataPool.m_safetyData.m_masterErrFlag[i] THEN
		m_nextMasterArmState[i] := MasterArmState_Error;
	END_IF
	
END_FOR

// To Endoscope Control 
IF SlaveArmState_ScopeReady = m_scopeArmState AND i_masterInputDataPool.m_cartStatus.m_endoscopeSwitch AND i_masterInputDataPool.m_cartStatus.m_surgonReady AND
  (MasterArmState_Standby = m_masterArmState[1] OR MasterArmState_Ready = m_masterArmState[1] OR MasterArmState_Matching = m_masterArmState[1] OR MasterArmState_MasterSlave = m_masterArmState[1]) AND 
  (MasterArmState_Standby = m_masterArmState[2] OR MasterArmState_Ready = m_masterArmState[2] OR MasterArmState_Matching = m_masterArmState[2] OR MasterArmState_MasterSlave = m_masterArmState[2]) THEN
	m_nextMasterArmState[1] := MasterArmState_Endoscope;
	m_nextMasterArmState[2] := MasterArmState_Endoscope;
END_IF
END_METHOD

METHOD PROTECTED updateShoulderPose : BOOL
VAR_INPUT
END_VAR
VAR
	monitorRot :mat3d;
END_VAR
// base monitor frame(0 rotation angle) in current monitor frame 
monitorRot := rotY( -m_monitorAngle);

// shoulder pose in current monitor frame
matMultiply(g_shoulderRotInMonitor,monitorRot, m_shoulderPoseInMonitor[1].m_rot);
m_shoulderPoseInMonitor[2].m_rot:=m_shoulderPoseInMonitor[1].m_rot;
END_METHOD

METHOD USKnifeClutchCheck : BOOL
VAR_IN_OUT CONSTANT
	i_masterInputDataPool:ST_MasterInputDataPool;
END_VAR

VAR
	i:INT;
END_VAR
FOR i:=1 TO g_sArmNum DO
	IF NOT(i_masterInputDataPool.m_slaveStatus.m_instruStauts[i].m_ready) THEN
		m_USKnifeRotClutch[i] := FALSE;
	END_IF
END_FOR

FOR i:=1 TO g_mArmNum DO
	IF (i_masterInputDataPool.m_slaveStatus.m_instruStauts[m_teleSlaveArmIdx[i]].m_type = InstruType_UltrasoundKnifeS OR i_masterInputDataPool.m_slaveStatus.m_instruStauts[m_teleSlaveArmIdx[i]].m_type = InstruType_UltrasoundKnifeU)
		AND  m_masterArmState[i] = MasterArmState_Clutch AND m_masterArms[i].handClutchSwitch THEN
		m_USKnifeRotClutch[m_teleSlaveArmIdx[i]] := TRUE;
	END_IF
END_FOR
END_METHOD

END_FUNCTION_BLOCK

// ---- FBs_Auxiliary/FB_slaveConnectionCheck.TcPOU
FUNCTION_BLOCK FB_slaveConnectionCheck
VAR
	// current state 
	m_isConnected :BOOL :=FALSE;
	
	// last heart beat
	m_lastHeartBeat :INT:=0 ;
	
	// current conneciton cycles
	m_curConnectionCycles :INT:=0;
	
	// current disconneciton cycles
	m_curDisconnectionCycles :INT:=0;
	
	// conneciton cycles thresshold
	m_connectionCyclesThres :INT:=5;
	
END_VAR

METHOD PUBLIC check : BOOL
VAR_INPUT
	i_heartBeat :INT;
END_VAR
// current is disconnected
IF NOT(m_isConnected) THEN
	m_curDisconnectionCycles:=0;
	
	IF  i_heartBeat <> m_lastHeartBeat THEN
		m_curConnectionCycles :=  m_curConnectionCycles +1;
	ELSE
		m_curConnectionCycles :=0;
	END_IF
	
	IF  m_curConnectionCycles >= m_connectionCyclesThres THEN
		m_isConnected := TRUE;
	END_IF

// current is connected
ELSE
	m_curConnectionCycles :=0;
	
	IF  i_heartBeat = m_lastHeartBeat THEN
		m_curDisconnectionCycles := m_curDisconnectionCycles +1;
	ELSE
		m_curDisconnectionCycles :=0;
	END_IF
	
	IF m_curDisconnectionCycles>= m_connectionCyclesThres THEN
		m_isConnected:=FALSE;
	END_IF

END_IF

m_lastHeartBeat:= i_heartBeat;
check:=m_isConnected;
END_METHOD

END_FUNCTION_BLOCK

// ---- FBs_Robots/FB_MasterArm.TcPOU
FUNCTION_BLOCK FB_MasterArm
VAR
	// arm index, 1 for left arm, 2 for right arm
	m_armIdx: INT;
	
	// grip angle calculator
	m_gripHallSensorIO AT%I* :UDINT;	
	m_gripAngleCalc : FB_GripAngleCalc;
	m_gripAngle :LREAL;
	
	//hand clutch switch IO
	m_handClutchIO AT%I*:UDINT;
	m_handClutchCheck :FB_HandClutchCheck;
	m_handClutchSwitch :BOOL;
	
	// joints
	// NOTICE: all joints are the true active joints, not DH ones!
	m_joints :ARRAY[1..g_mJntNum] OF FB_ArmJoint;
	
	// master gripper roll flip flag, if true, q7 would add pi in FK
	m_gripperRollFlip :BOOL :=False;
	
	// arm cartesian data, defined in each arm origin
	m_curCartPose	:ST_Frame;
	m_curCartTwist: Vec6d;
	m_cmdCartTwist :Vec6d;
	m_cmdCartPose:ST_Frame;
	m_curCartLinkPose :ST_Frame;
	m_curCartLinkTwist :Vec6d;
	
	
	// arm joint data
	m_curMotorPos :Vec7d;
	m_curLinkPos :Vec7d;
	m_curJntPos :Vec7d;
	m_curJntVel :Vec7d;
	m_curLinkVel :Vec7d;
	m_curJntTrq :Vec7d;
	m_rawJntCurrent :Vec7d;
	m_filtJntCurrent :Vec7d;
	m_cmdJntCurrent : Vec7d;
	m_cmdJntTrq :Vec7d;
	m_cmdJntPos :Vec7d;
	m_cmdJntVel :Vec7d;

	
	// arm dynamic data
	m_jntGravity : Vec7d;
	m_jntMassMat : Mat7d;
	m_lambda :Mat6d;
	m_dynaNullspace :Mat7d;
	m_jntFriction :Vec7d;
	m_jntExtTrq :Vec7d;
	
	// arm jacobian 
	m_jaco : Mat67;
	m_linkJaco : Mat67;
	
	// simulated status
	m_simJntPos :Vec7d;
	m_simCartPose : ST_Frame;
	m_simJaco : Mat67;
	
	// joint position controller
	m_jntPIDCtrl :ARRAY[1..g_mJntNum] OF FB_PID;
	
END_VAR

PROPERTY armIdx : int
GET
armIdx:=m_armIdx;
END_GET
END_PROPERTY

METHOD PROTECTED calcJaco : BOOL
VAR_IN_OUT CONSTANT
	i_jntPos :ARRAY[1..g_mJntNum] OF LREAL;
END_VAR
VAR_IN_OUT
	r_jaco :ARRAY[1..g_cartDofs, 1..g_mJntNum] OF LREAL;
END_VAR
VAR_INPUT
END_VAR

VAR
	q1,q2, q3, q4, q5, q6, q7 :LREAL;
	d1,d4,a3,a4 :LREAL;
	c1,c2,c3,c4,c5,c6,c7 :LREAL;
	s1,s2,s3,s4,s5,s6,s7 :LREAL;
	c23, s23 :LREAL;
	j:INT;
END_VAR
// !Convert active joint position to DH model for kinematic calculation
q1:=i_jntPos[1];  
q2:=i_jntPos[2];  
q3:=i_jntPos[3]-i_jntPos[2];  //q3=q8-q2
q4:=i_jntPos[4]+i_jntPos[3]-i_jntPos[2]-pi/2;//q4DH=q4motor+q8-q2-90;  
q5:=i_jntPos[5];  
q6:=i_jntPos[6];  
q7:=i_jntPos[7];  
d1:=g_d1;
d4:=g_d4;
a3:=g_a3;
a4:=g_a4;
c1:=COS(q1);
c2:=COS(q2);
c3:=COS(q3);
c4:=COS(q4);
c5:=COS(q5);
c6:=COS(q6);
c7:=COS(q7);
s1:=SIN(q1);
s2:=SIN(q2);
s3:=SIN(q3);
s4:=SIN(q4);
s5:=SIN(q5);
s6:=SIN(q6);
s7:=SIN(q7);
c23:=COS(q2+q3);
s23:=SIN(q2+q3);

// jacobian with DH joints
r_jaco[1,1]:=-s1*(c2*(a3 + a4*c3 - d4*s3) - s2*(d4*c3 + a4*s3)) ;
r_jaco[1,2]:=-c1*(s2*(a3 + a4*c3 - d4*s3) + c2*(d4*c3 + a4*s3)) ;
r_jaco[1,3]:=-c1*(d4*c23 + a4*s23) ;
r_jaco[1,4]:=0 ;
r_jaco[1,5]:=0 ;
r_jaco[1,6]:=0 ;
r_jaco[1,7]:=0;
 
r_jaco[2,1]:=c1*(c2*(a3 + a4*c3 - d4*s3) - s2*(d4*c3 + a4*s3)); 
r_jaco[2,2]:=-s1*(s2*(a3 + a4*c3 - d4*s3) + c2*(d4*c3 + a4*s3)); 
r_jaco[2,3]:=-s1*(d4*c23 + a4*s23); 
r_jaco[2,4]:=0; 
r_jaco[2,5]:=0; 
r_jaco[2,6]:=0; 
r_jaco[2,7]:=0;

 
r_jaco[3,1]:=0 ;
r_jaco[3,2]:=- c1*(c1*c2*(a3 + a4*c3 - d4*s3) - c1*s2*(d4*c3 + a4*s3)) - s1*(c2*s1*(a3 + a4*c3 - d4*s3) - s1*s2*(d4*c3 + a4*s3));
r_jaco[3,3]:=- c1*(a4*c23*c1 - d4*s23*c1) - s1*(a4*c23*s1 - d4*s23*s1);
r_jaco[3,4]:=0;
r_jaco[3,5]:=0;
r_jaco[3,6]:=0 ;
r_jaco[3,7]:=0 ;

r_jaco[4,1]:=0 ;
r_jaco[4,2]:=-s1 ;
r_jaco[4,3]:=-s1 ;
r_jaco[4,4]:=-s23*c1 ;
r_jaco[4,5]:=c23*c1*s4 - c4*s1 ;
r_jaco[4,6]:=- s5*(s1*s4 + c23*c1*c4) - s23*c1*c5 ;
r_jaco[4,7]:=s6*(c5*(s1*s4 + c4*(c1*c2*c3 - c1*s2*s3)) - s5*(c1*c2*s3 + c1*c3*s2)) - c6*(c4*s1 - s4*(c1*c2*c3 - c1*s2*s3));
 
r_jaco[5,1]:=0; 
r_jaco[5,2]:=c1; 
r_jaco[5,3]:=c1; 
r_jaco[5,4]:=-s23*s1; 
r_jaco[5,5]:=c1*c4 + c23*s1*s4; 
r_jaco[5,6]:=s5*(c1*s4 - c23*c4*s1) - s23*c5*s1; 
r_jaco[5,7]:=c6*(c1*c4 - s4*(s1*s2*s3 - c2*c3*s1)) - s6*(c5*(c1*s4 + c4*(s1*s2*s3 - c2*c3*s1)) + s5*(c2*s1*s3 + c3*s1*s2));

r_jaco[6,1]:=1 ;
r_jaco[6,2]:=0 ;
r_jaco[6,3]:=0 ;
r_jaco[6,4]:=-c23 ;
r_jaco[6,5]:=-s23*s4 ;
r_jaco[6,6]:=s23*c4*s5 - c23*c5 ;
r_jaco[6,7]:=- s6*(c23*s5 + s23*c4*c5) - s23*c6*s4;

// jacobian with active joints
// jaco_DH*qdot_DH = jaco_DH * (A * qdot)= jaco * qdot
// A =[ 1  0 0 0 0 0 0
//		0  1 0 0 0 0 0
//		0 -1 1 0 0 0 0
//		0 -1 1 1 0 0 0
//		0 0  0 0 1 0 0
//      0 0  0 0 0 1 0
// 		0 0  0 0 0 0 1]
 FOR j:=1 TO 6 DO 
	 r_jaco[j,2]:=r_jaco[j,2]-r_jaco[j,3]-r_jaco[j,4];
	 r_jaco[j,3]:=r_jaco[j,3]+r_jaco[j,4];
 END_FOR
END_METHOD

PROPERTY cmdCartPose : REFERENCE TO ST_Frame
GET
cmdCartPose REF= m_cmdCartPose;
END_GET
END_PROPERTY

PROPERTY cmdCartTwist : REFERENCE to Vec6d
GET
cmdCartTwist REF= m_cmdCartTwist;
END_GET
END_PROPERTY

PROPERTY cmdJntCurrent :REFERENCE to Vec7d
GET
cmdJntCurrent REF= m_cmdJntCurrent;
END_GET
END_PROPERTY

PROPERTY cmdJntPos : REFERENCE TO Vec7d
GET
cmdJntPos REF= m_cmdJntPos;
END_GET
END_PROPERTY

PROPERTY cmdJntTrq :REFERENCE TO Vec7d
GET
cmdJntTrq REF= m_cmdJntTrq;
END_GET
END_PROPERTY

PROPERTY cmdJntVel : REFERENCE TO Vec7d
GET
cmdJntVel REF= m_cmdJntVel;
END_GET
END_PROPERTY

PROPERTY curCartPose :REFERENCE to ST_Frame
GET
curCartPose REF=m_curCartPose;
END_GET
END_PROPERTY

PROPERTY curCartTwist :REFERENCE TO Vec6d
GET
curCartTwist REF=m_curCartTwist;
END_GET
END_PROPERTY

PROPERTY curJntPos :REFERENCE TO Vec7d
GET
curJntPos REF=m_curJntPos;
END_GET
END_PROPERTY

PROPERTY curJntTrq :REFERENCE TO Vec7d
GET
curJntTrq REF=m_curJntTrq;
END_GET
END_PROPERTY

PROPERTY curJntVel :REFERENCE TO Vec7d
GET
curJntVel REF=m_curJntVel;
END_GET
END_PROPERTY

PROPERTY curLinkPos :REFERENCE TO  Vec7d
GET
curLinkPos REF=m_curLinkPos;
END_GET
END_PROPERTY

PROPERTY curMotorPos :REFERENCE TO Vec7d
GET
curMotorPos REF=m_curMotorPos;
END_GET
END_PROPERTY

PROPERTY PUBLIC dynaNullspace : REFERENCE TO Mat7d
GET
dynaNullspace REF= m_dynaNullspace;
END_GET
END_PROPERTY

METHOD PROTECTED enable : BOOL
VAR_IN_OUT CONSTANT
	i_jntIdx :Vec7i;
END_VAR
VAR
	i :INT ;
END_VAR
FOR i:=1 TO g_mJntNum DO
	IF 1= i_jntIdx[i] THEN
		m_joints[i].enable();
	ELSE
		m_joints[i].disable();
	END_IF
END_FOR
END_METHOD

PROPERTY filtJntCurrent :REFERENCE to Vec7d
GET
filtJntCurrent ref= m_filtJntCurrent;
END_GET
END_PROPERTY

METHOD PUBLIC flipGripper : BOOL
VAR_INPUT
	i_flipFlag :BOOL;
END_VAR
m_gripperRollFlip := i_flipFlag;
END_METHOD

// from active joint position to cartesian pose in arm origin
METHOD PROTECTED forwardKinematic : BOOL
VAR_IN_OUT CONSTANT
	i_jntPos :ARRAY[1..g_mJntNum] OF LREAL;
END_VAR
VAR_IN_OUT
	r_cartPose :ST_Frame;
END_VAR
VAR
	q1,q2, q3, q4, q5, q6, q7 :LREAL;
	d1,d4,a3,a4 :LREAL;
	c1,c2,c3,c4,c5,c6,c7 :LREAL;
	s1,s2,s3,s4,s5,s6,s7 :LREAL;
	c23, s23 :LREAL;
END_VAR
// !Convert active joint position to DH model for kinematic calculation
q1:=i_jntPos[1];  
q2:=i_jntPos[2];  
q3:=i_jntPos[3]-i_jntPos[2];  //q3=q8-q2
q4:=jnt4MotorToLink(i_jntPos[2],i_jntPos[3], i_jntPos[4]);//q4DH=q4motor+q8-q2-90;  
q5:=i_jntPos[5];  
q6:=i_jntPos[6];  
q7:=i_jntPos[7];  

// master roll flip handle
IF m_gripperRollFlip THEN
	q7 := q7+PI;
END_IF

d1:=g_d1;
d4:=g_d4;
a3:=g_a3;
a4:=g_a4;
c1:=COS(q1);
c2:=COS(q2);
c3:=COS(q3);
c4:=COS(q4);
c5:=COS(q5);
c6:=COS(q6);
c7:=COS(q7);
s1:=SIN(q1);
s2:=SIN(q2);
s3:=SIN(q3);
s4:=SIN(q4);
s5:=SIN(q5);
s6:=SIN(q6);
s7:=SIN(q7);
c23:=COS(q2+q3);
s23:=SIN(q2+q3);

// cartesian pose frame
r_cartPose.m_pos[1]:=c1*(a4*c23 - d4*s23 + a3*c2); 
r_cartPose.m_pos[2]:=s1*(a4*c23 - d4*s23 + a3*c2);
r_cartPose.m_pos[3]:=d1 - d4*c23 - a4*s23 - a3*s2;  
r_cartPose.m_rot[1,1]:=c7*(s6*(c4*s1 - s4*(c1*c2*c3 - c1*s2*s3)) + c6*(c5*(s1*s4 + c4*(c1*c2*c3 - c1*s2*s3)) - s5*(c1*c2*s3 + c1*c3*s2))) - s7*(s5*(s1*s4 + c4*(c1*c2*c3 - c1*s2*s3)) + c5*(c1*c2*s3 + c1*c3*s2));
r_cartPose.m_rot[2,1]:=s7*(s5*(c1*s4 + c4*(s1*s2*s3 - c2*c3*s1)) - c5*(c2*s1*s3 + c3*s1*s2)) - c7*(s6*(c1*c4 - s4*(s1*s2*s3 - c2*c3*s1)) + c6*(c5*(c1*s4 + c4*(s1*s2*s3 - c2*c3*s1)) + s5*(c2*s1*s3 + c3*s1*s2)));
r_cartPose.m_rot[3,1]:=- s7*(c23*c5 - s23*c4*s5) - c7*(c23*c6*s5 - s23*s4*s6 + s23*c4*c5*c6); 
r_cartPose.m_rot[1,2]:=- s7*(s6*(c4*s1 - s4*(c1*c2*c3 - c1*s2*s3)) + c6*(c5*(s1*s4 + c4*(c1*c2*c3 - c1*s2*s3)) - s5*(c1*c2*s3 + c1*c3*s2))) - c7*(s5*(s1*s4 + c4*(c1*c2*c3 - c1*s2*s3)) + c5*(c1*c2*s3 + c1*c3*s2)); 
r_cartPose.m_rot[2,2]:=s7*(s6*(c1*c4 - s4*(s1*s2*s3 - c2*c3*s1)) + c6*(c5*(c1*s4 + c4*(s1*s2*s3 - c2*c3*s1)) + s5*(c2*s1*s3 + c3*s1*s2))) + c7*(s5*(c1*s4 + c4*(s1*s2*s3 - c2*c3*s1)) - c5*(c2*s1*s3 + c3*s1*s2)); 
r_cartPose.m_rot[3,2]:=s7*(c23*c6*s5 - s23*s4*s6 + s23*c4*c5*c6) - c7*(c23*c5 - s23*c4*s5); 
r_cartPose.m_rot[1,3]:=s6*(c5*(s1*s4 + c4*(c1*c2*c3 - c1*s2*s3)) - s5*(c1*c2*s3 + c1*c3*s2)) - c6*(c4*s1 - s4*(c1*c2*c3 - c1*s2*s3)); 
r_cartPose.m_rot[2,3]:=c6*(c1*c4 - s4*(s1*s2*s3 - c2*c3*s1)) - s6*(c5*(c1*s4 + c4*(s1*s2*s3 - c2*c3*s1)) + s5*(c2*s1*s3 + c3*s1*s2));
r_cartPose.m_rot[3,3]:=- s6*(c23*s5 + s23*c4*c5) - s23*c6*s4;
END_METHOD

PROPERTY gripAngle : LREAL
GET
gripAngle:=m_gripAngle;
END_GET
END_PROPERTY

PROPERTY gripperRollFlip : BOOL
GET
gripperRollFlip := m_gripperRollFlip;
END_GET
END_PROPERTY

PROPERTY handClutchSwitch : BOOL
GET
handClutchSwitch :=m_handClutchSwitch;
END_GET
END_PROPERTY

METHOD PUBLIC init : BOOL
VAR_INPUT
	i_armIdx:INT;
END_VAR
VAR 
	i :INT ;
	currentRatioMotor2Jnt: LREAL;
END_VAR
// arm statues init
m_armIdx:=i_armIdx;
m_gripAngle:=0;
m_gripAngleCalc.init(m_armIdx);

// joint init
FOR i:=1 TO g_mJntNum DO
	m_joints[i].init(m_armIdx, i,g_armCtrlCycleTime);
END_FOR

// init joint encoder and position calculation
initJntPos();

// joint controller init
FOR i:=1 TO g_mJntNum DO 
	currentRatioMotor2Jnt:=GVL_ArmJointParameters.g_motorTrqConst[i]*GVL_ArmJointParameters.g_motorReduction[i]/1000;
	m_jntPIDCtrl[i].init(g_armCtrlCycleTime,g_posKp[i],g_posKd[i],g_posKi[i],
		g_posKiLimit[i]* currentRatioMotor2Jnt,	g_posCtrlLimit[i]*currentRatioMotor2Jnt);
END_FOR
END_METHOD

METHOD public initJntPos : BOOL
VAR_INPUT
END_VAR
VAR
	i:INT ;
	initLinkPos:LREAL;
END_VAR
// joint init
FOR i:=1 TO g_mJntNum DO
	m_joints[i].initJntPos();
END_FOR

// link position of joint4 is influenced by joint2 and joint3, need to handle seperately
initLinkPos:=jnt4LinkToMotor(m_joints[2].initLinkPos,m_joints[3].initLinkPos, m_joints[4].initLinkPos);
m_joints[4].initJntPosReset(initLinkPos);

// update arm status after joint position is re-init
updateStatus();
END_METHOD

// from cartesian pose in arm origin to active joint position
METHOD PROTECTED inverseKinematic : BOOL
VAR_INPUT
	q4:LREAL;
	solution_ID:INT;
END_VAR
VAR_IN_OUT CONSTANT
	i_curCartPose :ST_Frame;
END_VAR
VAR_IN_OUT
	r_jntPos :ARRAY[1..g_mJntNum] OF LREAL;
END_VAR
VAR
	a3,a4,d1,d4:LREAL;
	px,py,pz:lreal;
	nx,ny,nz:lreal;
	ox,oy,oz:lreal;
	ax,ay,az:lreal;

	q1,q2,q3,q5,q6,q7:LREAL;
	
	q11,q12:LREAL;
	k1,A,B,C,fi,R0,q21,q22:lreal;
	ins1,ins2:lreal;
	
	A11,A12,A21,A22,C1,C2:lreal;
	SIN23,COS23,q23:lreal;
	
	T_74_left_23,q61,q62:lreal;
	T_74_left_13,T_74_left_33:lreal;
	T_74_left_21,T_74_left_22:LREAL;	
	
	succeed_1,succeed_2,succeed:BOOL;
END_VAR


//***********************单臂逆向运动学**************************//
d1:=g_d1;
d4:=g_d4;
a3:=g_a3;
a4:=g_a4;

nx:=i_curCartPose.m_rot[1,1];  ny:=i_curCartPose.m_rot[2,1];  nz:=i_curCartPose.m_rot[3,1];
ox:=i_curCartPose.m_rot[1,2]; oy:=i_curCartPose.m_rot[2,2];  oz:=i_curCartPose.m_rot[3,2];
ax:=i_curCartPose.m_rot[1,3];  ay:=i_curCartPose.m_rot[2,3];  az:=i_curCartPose.m_rot[3,3];
px:=i_curCartPose.m_pos[1]; py:=i_curCartPose.m_pos[2]; pz:=i_curCartPose.m_pos[3];


//求解q1
q11:=atan2(y:= py, x:= px);
q12:=-q11;
IF (Solution_ID<=4) THEN
	q1:=q11;
ELSE
	q1:=q12;
END_IF



//求解q2
k1:=px*COS(q1) + py*SIN(q1);
A:=2*a3*pz - 2*a3*d1;
B:=2*a3*k1;
C:=a3*a3 - a4*a4 + d1*d1 - 2*d1*pz - d4*d4 + k1*k1 + pz*pz;
fi:=atan2(y:= B, x:= A);

R0:=SQRT(A*A+B*B);

//*************程序保护性处理，避免软件崩溃***************//
IF ABS(C/R0)>1 THEN
	succeed_1:=FALSE;
	succeed:=FALSE;
	RETURN;
ELSE
	succeed_1:=TRUE;
END_IF

ins1:=atan2(y:= C/R0, x:= SQRT(1-(C/R0)*(C/R0)));
q21:=fi-ins1;
ins2:=atan2(y:= C/R0, x:= -SQRT(1-(C/R0)*(C/R0)));
q22:=fi-ins2;

IF (Solution_ID=1) OR (Solution_ID=2) OR (Solution_ID=5) OR (Solution_ID=6) THEN
	q2:=q21;
ELSE
	q2:=q22;
END_IF




//求解q3
A11:=- d4;
A12:=a4;
A21:=- a4;
A22:=-d4;
C1:=k1- a3*COS(q2);
C2:=pz - d1 + a3*SIN(q2);
sin23:=(C1*A22-C2*A12)/(A11*A22-A21*A12);
cos23:=(C2*A11-C1*A21)/(A11*A22-A21*A12);
q23:=atan2(y:= sin23, x:= cos23);
q3:=q23-q2;




//求解q6
T_74_left_23:=ax*(COS(q4)*SIN(q1) - COS(q1)*COS(q2)*COS(q3)*SIN(q4) + COS(q1)*SIN(q2)*SIN(q3)*SIN(q4)) - ay*(COS(q1)*COS(q4) + COS(q2)*COS(q3)*SIN(q1)*SIN(q4) - SIN(q1)*SIN(q2)*SIN(q3)*SIN(q4)) + az*SIN(q2 + q3)*SIN(q4);

//*************程序保护性处理，避免软件崩溃***************//
IF ABS(T_74_left_23>1) THEN
	succeed_2:=FALSE;
	succeed:=FALSE;
	RETURN;
ELSE
	succeed_2:=TRUE;
END_IF

q61:=ACOS(-T_74_left_23);
q62:=-ACOS(-T_74_left_23);
IF (Solution_ID=1) OR (Solution_ID=3) OR (Solution_ID=5) OR (Solution_ID=7) THEN
	q6:=q61;
ELSE
	q6:=q62;
END_IF


//求解q5
T_74_left_13:=ax*(SIN(q1)*SIN(q4) + COS(q1)*COS(q2)*COS(q3)*COS(q4) - COS(q1)*COS(q4)*SIN(q2)*SIN(q3)) - ay*(COS(q1)*SIN(q4) - COS(q2)*COS(q3)*COS(q4)*SIN(q1) + COS(q4)*SIN(q1)*SIN(q2)*SIN(q3)) - az*SIN(q2 + q3)*COS(q4);
T_74_left_33:=- az*COS(q2 + q3) - ax*SIN(q2 + q3)*COS(q1) - ay*SIN(q2 + q3)*SIN(q1);
q5:=atan2(y:= T_74_left_33*SIN(q6), x:= T_74_left_13*SIN(q6));


//求解q7
T_74_left_21:=nx*(COS(q4)*SIN(q1) - COS(q1)*COS(q2)*COS(q3)*SIN(q4) + COS(q1)*SIN(q2)*SIN(q3)*SIN(q4)) - ny*(COS(q1)*COS(q4) + COS(q2)*COS(q3)*SIN(q1)*SIN(q4) - SIN(q1)*SIN(q2)*SIN(q3)*SIN(q4)) + nz*SIN(q2 + q3)*SIN(q4);
T_74_left_22:=ox*(COS(q4)*SIN(q1) - COS(q1)*COS(q2)*COS(q3)*SIN(q4) + COS(q1)*SIN(q2)*SIN(q3)*SIN(q4)) - oy*(COS(q1)*COS(q4) + COS(q2)*COS(q3)*SIN(q1)*SIN(q4) - SIN(q1)*SIN(q2)*SIN(q3)*SIN(q4)) + oz*SIN(q2 + q3)*SIN(q4);
q7:=atan2(y:= -T_74_left_22*SIN(q6), x:= T_74_left_21*SIN(q6));


//! convert DH joint postion to active joint position
r_jntPos[1]:=q1;
r_jntPos[2]:=q2;
r_jntPos[3]:=q3+q2; // q8 = q3+q2
r_jntPos[4]:=q4+q2-r_jntPos[3]+pi/2;//q4DH=q4motor+q8-q2-90;  
r_jntPos[5]:=q5;
r_jntPos[6]:=q6;
r_jntPos[7]:=q7;

succeed:=TRUE;
inverseKinematic:=succeed;
END_METHOD

METHOD PUBLIC isEnabled : BOOL
VAR_IN_OUT CONSTANT
	i_jntIdx :Vec7i;
END_VAR
VAR
	i :INT ;
END_VAR
isEnabled := TRUE;
FOR i:=1 TO g_mJntNum DO
	IF 1= i_jntIdx[i] THEN
		isEnabled :=  (m_joints[i].isEnabled() AND isEnabled);
	END_IF
END_FOR
END_METHOD

PROPERTY jaco :REFERENCE to Mat67
GET
jaco ref= m_jaco;
END_GET
END_PROPERTY

//convert joint4 position from link side to motor side
METHOD PUBLIC jnt4LinkToMotor : LREAL
VAR_INPUT
	i_q2 :LREAL;
	i_q3:LREAL;
	i_q4Link :LREAL;
END_VAR
jnt4LinkToMotor:=i_q4Link-i_q3+i_q2+pi/2;//q4motor=q4DH-q8+q2+90;
END_METHOD

//convert joint4 position from motor side to link side
METHOD public jnt4MotorToLink : LREAL
VAR_INPUT
	i_q2 :LREAL;
	i_q3:LREAL;
	i_q4Motor :LREAL;
END_VAR
jnt4MotorToLink:=i_q4Motor+i_q3-i_q2-pi/2;//q4DH=q4motor+q8-q2-90;
END_METHOD

PROPERTY jntExtTrq :REFERENCE TO Vec7d
GET
jntExtTrq REF= m_jntExtTrq;
END_GET
END_PROPERTY

PROPERTY jntFriction :REFERENCE TO Vec7d
GET
jntFriction REF= m_jntFriction;
END_GET
END_PROPERTY

PROPERTY jntGravity :REFERENCE to Vec7d
GET
jntGravity ref=m_jntGravity;
END_GET
END_PROPERTY

PROPERTY PUBLIC massMat :REFERENCE to Mat7d
GET
massMat ref=m_jntMassMat;
END_GET
END_PROPERTY

PROPERTY rawJntCurrent :REFERENCE to Vec7d
GET
rawJntCurrent ref=m_rawJntCurrent;
END_GET
END_PROPERTY

PROPERTY simCartPose :REFERENCE to ST_Frame
GET
simCartPose REF=m_simCartPose;
END_GET
END_PROPERTY

PROPERTY simJaco :REFERENCE TO mat67
GET
simJaco REF=m_simJaco;
END_GET
END_PROPERTY

// update joints control command
METHOD PUBLIC updateCmds : BOOL
VAR_IN_OUT CONSTANT
	i_armCtrlCmd : ST_ArmCtrlCmds;
END_VAR
VAR
	i:INT;
END_VAR
m_cmdJntTrq:=i_armCtrlCmd.m_cmdJntTrq;
m_cmdJntPos :=i_armCtrlCmd.m_cmdJntPos;
m_cmdJntVel :=i_armCtrlCmd.m_cmdJntVel;
m_cmdCartTwist := i_armCtrlCmd.m_cmdCartTwist;
m_cmdCartPose :=i_armCtrlCmd.m_cmdCartPose;
m_simJntPos:=i_armCtrlCmd.m_cmdJntPos;

// update simulated master arm
updateSimStatus();

// enable/disable joints
enable(i_armCtrlCmd.m_jntEnableFlag);

// position/torque control
FOR i:=1 TO g_mJntNum DO 
	IF i_armCtrlCmd.m_jntOPMode[i]=DriverOPMode_PosTrq THEN
		// position controller and gravity feedforward
		m_cmdJntTrq[i]:=m_jntPIDCtrl[i].run(i_armCtrlCmd.m_cmdJntPos[i],m_curJntPos[i],i_armCtrlCmd.m_cmdJntVel[i],m_curJntVel[i]);
		m_cmdJntTrq[i]:=m_cmdJntTrq[i]+m_jntGravity[i];
		m_joints[i].updateCmds(DriverOPMode_Trq,i_armCtrlCmd.m_cmdJntPos[i],m_cmdJntTrq[i]);
	ELSIF i_armCtrlCmd.m_jntOPMode[i]=DriverOPMode_Trq THEN
		// gravity feedforward
		m_jntPIDCtrl[i].reset();
		m_cmdJntTrq[i]:=m_cmdJntTrq[i]+m_jntGravity[i];
		m_joints[i].updateCmds(DriverOPMode_Trq,i_armCtrlCmd.m_cmdJntPos[i],m_cmdJntTrq[i]);
	ELSE
		m_jntPIDCtrl[i].reset();
		m_cmdJntTrq[i]:=0;
		m_joints[i].updateCmds(DriverOPMode_Pos,i_armCtrlCmd.m_cmdJntPos[i],m_cmdJntTrq[i]);
	END_IF
	
END_FOR
END_METHOD

METHOD PUBLIC updateDyna : BOOL
VAR_IN_out constant
	masterDynaData : ST_MasterDynaData;
END_VAR
m_jntMassMat:=masterDynaData.m_massMat[m_armIdx];
m_lambda:=masterDynaData.m_lambda[m_armIdx];
m_dynaNullspace:=masterDynaData.m_dynaNullspace[m_armIdx];
m_jntGravity:=masterDynaData.m_gravity[m_armIdx];
m_jntFriction:=masterDynaData.m_friction[m_armIdx];
m_jntExtTrq := masterDynaData.m_jntExtTrq[m_armIdx];
END_METHOD

METHOD PUBLIC updateSimStatus : BOOL
VAR_INPUT
END_VAR
// simulated cartesion pose 
forwardKinematic(m_simJntPos,m_simCartPose);

// simulated jacobian
calcJaco(m_simJntPos,m_simJaco);
END_METHOD

// update arm status, including kinematic and dynamic
METHOD PUBLIC updateStatus : BOOL
VAR_INPUT
END_VAR
VAR 
	i,j:INT;
END_VAR
// grip angle
m_gripAngle :=m_gripAngleCalc.run(m_gripHallSensorIO);

// check hand clutch
m_handClutchSwitch :=  m_handClutchCheck.run(m_handClutchIO);

// update joint data
FOR i:=1 TO g_mJntNum DO
	m_joints[i].updateStatus();
END_FOR

// get joint data
FOR i:=1 TO g_mJntNum DO
	m_curMotorPos[i]:=m_joints[i].motorPos;
	m_curLinkPos[i]:=m_joints[i].linkPos;
	m_curJntPos[i]:=m_joints[i].jntPos;
	m_curJntVel[i]:=m_joints[i].jntVel;
	m_curLinkVel[i] := m_joints[i].m_curLinkVel;
	m_curJntTrq[i]:=m_joints[i].jntTrq;
	m_rawJntCurrent[i]:=m_joints[i].rawCurrent;
	m_filtJntCurrent[i]:=m_joints[i].filtCurrent;
	m_cmdJntCurrent[i]:=m_joints[i].cmdCurrent;
END_FOR 
m_curLinkPos[4]:=jnt4LinkToMotor(m_curLinkPos[2],m_curLinkPos[3], m_curLinkPos[4]);// q4motor=q4DH-q8+q2+90; 
m_curLinkVel[4]:= m_curLinkVel[4] - m_curLinkVel[3] + m_curLinkVel[2]; 

// cartesion pose
forwardKinematic(m_curJntPos,m_curCartPose);
forwardKinematic(m_curLinkPos,m_curCartLinkPose);

// jacobian
calcJaco(m_curJntPos,m_jaco);
calcJaco(m_curLinkPos,m_linkJaco);

// cartesian twist
matMultiVec(m_jaco,m_curJntVel,m_curCartTwist);
matMultiVec(m_linkJaco,m_curLinkVel,m_curCartLinkTwist);
END_METHOD

END_FUNCTION_BLOCK

// ---- FBs_Auxiliary/FB_GripAngleCalc.TcPOU
FUNCTION_BLOCK FB_GripAngleCalc
VAR_INPUT
END_VAR
VAR_OUTPUT
END_VAR
VAR
	// limit value
	m_minHallSensorValue :LREAL;
	m_maxHallSensorValue:LREAL;
	m_hallSensorRange:LREAL;
	
	// grip angle from hall sensor IO
	m_gripHallSenorValue :LREAL;
	m_normHallSensorValue: LREAL;
	m_gripAngle :LREAL;
	m_gripAngLpf : FB_LowPassFilter;
END_VAR

METHOD init : BOOL
VAR_INPUT
	i_armIdx:INT;
END_VAR
// init limit value
m_minHallSensorValue:=(GVL_ArmJointCaliData.g_minHallSensorValue[i_armIdx]/65536) AND 16#0000FFFF; 
m_maxHallSensorValue:=(GVL_ArmJointCaliData.g_maxHallSensorValue[i_armIdx]/65536) AND 16#0000FFFF; 
m_hallSensorRange := m_maxHallSensorValue-m_minHallSensorValue;

// init filter
m_gripAngLpf.init(1, g_gripAngLpfCutoffFreq, g_armCtrlFreq);
END_METHOD

METHOD run : LREAL
VAR_INPUT
	IOValue : UDINT;
END_VAR
// sensor io parse
m_gripHallSenorValue:=(IOValue/65536) AND 16#0000FFFF; //high 16 bits

// normalize hall sensor value
m_normHallSensorValue:=LIMIT(0, (m_gripHallSenorValue-m_minHallSensorValue)/m_hallSensorRange, 1);

// grip angle fitting
m_gripAngle := g_masterGripAngleFitCoeff[1] * EXPT(m_normHallSensorValue,5)
			+ g_masterGripAngleFitCoeff[2] * EXPT(m_normHallSensorValue,4)
			+ g_masterGripAngleFitCoeff[3] * EXPT(m_normHallSensorValue,3)
			+ g_masterGripAngleFitCoeff[4] * EXPT(m_normHallSensorValue,2)
			+ g_masterGripAngleFitCoeff[5] * EXPT(m_normHallSensorValue,1)
			+ g_masterGripAngleFitCoeff[6];
	
// filt and cap the result
m_gripAngle := m_gripAngLpf.run(m_gripAngle);
m_gripAngle := LIMIT(g_minGripAngle, m_gripAngle, g_maxGripAngle);

run:=m_gripAngle;
END_METHOD

END_FUNCTION_BLOCK

// ---- FBs_Filters/FB_LowPassFilter.TcPOU
// Low pass filter based on tusin transformation
// Author: Ni Feijian
// Data: 2023.11.27
FUNCTION_BLOCK FB_LowPassFilter
VAR_INPUT
END_VAR
VAR_OUTPUT
END_VAR
VAR
	// first data flag
	m_firstData:BOOL:=true;
	
	// sample frequency
	m_sampleFreq:LREAL;
	
	// cutoff frequency
	m_cutoffFreq:LREAL;
	
	// filter order
	m_filterOrd:INT:=1;
	
	// historic input data
	m_xk_1:LREAL;
	
	// coefficient for  input data
	m_cxk_1: LREAL;
	
	// historic output data
	m_yk_1:LREAL;
	
	// coefficient for output data
	m_cyk_1:LREAL;
END_VAR

METHOD PUBLIC init : BOOL
VAR_INPUT
	// filter orde
	i_filterOrd:INT;
	
	// cutoff frequency
	i_cutoffFreq:LREAL;
	
	// sample frequency
	i_sampleFreq:LREAL;
END_VAR
VAR
	tgw:LREAL;
END_VAR
m_firstData:=TRUE;
m_filterOrd:=1; // we currenty support fisrt order filt
m_cutoffFreq:=i_cutoffFreq;
m_sampleFreq:=i_sampleFreq;

CASE m_filterOrd OF
1:
	tgw:=TAN(pi*m_cutoffFreq/m_sampleFreq);
	m_cxk_1:=tgw/(tgw+1);
	m_cyk_1:=(tgw-1)/(tgw+1);
	init:=TRUE;
ELSE
	init :=FALSE;
END_CASE
END_METHOD

METHOD reset : BOOL
VAR_INPUT
END_VAR
m_firstData:=true;
END_METHOD

METHOD PUBLIC run : LREAL
VAR_INPUT
	// raw data
	i_rawData:LREAL;
END_VAR
CASE m_filterOrd OF
1:
	IF m_firstData=TRUE THEN
		m_xk_1:=i_rawData;
		m_yk_1:=i_rawData;
		run:=i_rawData;
		m_firstData:=FALSE;
	ELSE
		run:= m_cxk_1*(i_rawData+m_xk_1)-m_cyk_1*m_yk_1;
		m_xk_1:=i_rawData;
		m_yk_1:=run;
	END_IF
ELSE
	run:=i_rawData;
END_CASE
END_METHOD

END_FUNCTION_BLOCK

// ---- FBs_Auxiliary/FB_HandClutchCheck.TcPOU
FUNCTION_BLOCK FB_HandClutchCheck
VAR_INPUT
END_VAR
VAR_OUTPUT
END_VAR
VAR
	m_handClutchSwitch :BOOL;
	m_handClutchOnCounts :INT;
	m_handClutchOnCountThres :INT :=50;
END_VAR

METHOD run : BOOL
VAR_INPUT
	IOValue :UDINT;
END_VAR
// TODO: The two hand clutch switch is mapped to 1/2 bits, but the IO value would change to 28 sometimes
//IF (IOValue AND 10#3) > 0 THEN
IF IOValue > 0 THEN
	m_handClutchOnCounts := MIN(m_handClutchOnCounts +1, m_handClutchOnCountThres);
ELSE
	 m_handClutchOnCounts :=0;
END_IF

m_handClutchSwitch:=m_handClutchOnCounts>=m_handClutchOnCountThres;
run:=m_handClutchSwitch;
END_METHOD

END_FUNCTION_BLOCK

// ---- FBs_Robots/FB_ArmJoint.TcPOU
FUNCTION_BLOCK FB_ArmJoint EXTENDS FB_JointBase
VAR_INPUT
END_VAR
VAR_OUTPUT
END_VAR
VAR
END_VAR

METHOD PUBLIC init : BOOL
VAR_INPUT
	i_armIdx :INT;
	i_jntIdx :INT;
	i_controlCycleTime :LREAL;
END_VAR
m_cycleTime := i_controlCycleTime;

// hardware parameters
m_motorEncoderRes :=GVL_ArmJointParameters.g_incEncoderRes[i_jntIdx];
m_linkEncoderRes :=GVL_ArmJointParameters.g_absEncoderRes[i_jntIdx];
m_motorReduction :=GVL_ArmJointParameters.g_motorReduction[i_jntIdx];
m_linkEncoderReduction :=GVL_ArmJointParameters.g_absEncoderReduction[i_jntIdx];
m_trqConst :=GVL_ArmJointParameters.g_motorTrqConst[i_jntIdx];
m_maxCurrent :=GVL_ArmJointParameters.g_motorMaxCurrent[i_jntIdx];
m_motorDir :=GVL_ArmJointParameters.g_motorDir[i_armIdx,i_jntIdx];								
m_linkEncoderDir :=GVL_ArmJointParameters.g_asbEncoderDir[i_armIdx,i_jntIdx];
m_minJntPos	:=GVL_ArmJointParameters.g_minJntPos[i_armIdx,i_jntIdx];
m_maxJntPos	:=GVL_ArmJointParameters.g_maxJntPos[i_armIdx,i_jntIdx];

//link encoder calibartion data
m_minLinkEncoder :=GVL_ArmJointCaliData.g_minLinkEncoder[i_armIdx, i_jntIdx] - m_linkEncoderDir*GVL_ArmJointCaliData.g_linkEncLimitBuffer; // expand limit
m_maxLinkEncoder :=GVL_ArmJointCaliData.g_maxLinkEncoder[i_armIdx, i_jntIdx] + m_linkEncoderDir*GVL_ArmJointCaliData.g_linkEncLimitBuffer; // expand limit
m_caliLinkEncoder :=GVL_ArmJointCaliData.g_caliLinkEncoder[i_armIdx, i_jntIdx];
m_linkEncCaliJntPos :=GVL_ArmJointCaliData.g_linkEncCaliJntPos[i_armIdx, i_jntIdx];
m_linkEncZeroCross :=GVL_ArmJointCaliData.g_linkEncZeroCross[i_armIdx, i_jntIdx];
m_multiCycles :=GVL_ArmJointCaliData.g_multipleCyclesJoint[i_armIdx,i_jntIdx];

// convert cali link encoder if joint cross zero
IF 1=m_linkEncZeroCross THEN
	IF 1=m_linkEncoderDir AND m_caliLinkEncoder < m_minLinkEncoder THEN
		m_caliLinkEncoder := GVL_ArmJointCaliData.g_caliLinkEncoder[i_armIdx, i_jntIdx] + m_linkEncoderRes;
	ELSIF -1=m_linkEncoderDir AND m_caliLinkEncoder < m_maxLinkEncoder THEN
		m_caliLinkEncoder := GVL_ArmJointCaliData.g_caliLinkEncoder[i_armIdx, i_jntIdx] + m_linkEncoderRes;
	END_IF
END_IF

// macro data
m_trq2CurrentRatio:=m_motorDir * 1000.0/(m_trqConst*m_motorReduction);
m_current2TrqRatio:=m_motorDir * (m_trqConst*m_motorReduction)/1000.0;
m_linkEnc2PosRatio := 2*PI*m_linkEncoderDir/(m_linkEncoderReduction*m_linkEncoderRes);
m_motorEnc2PosRatio := 2*PI * m_motorDir/(m_motorReduction * m_motorEncoderRes);

// motor data init
m_curJntVel:=0;
m_curJntTrq :=0;
m_rawCurrent :=0;
m_filtCurrent :=0;
m_cmdJntVel :=0.0;
m_cmdJntTrq :=0.0;
m_cmdCurrent := 0.0;

// filter init
m_jntVelLpf.init(1, g_curJntVelLpfCutoffFreq, g_armCtrlFreq);
m_linkVelLpf.init(1, g_curJntVelLpfCutoffFreq, g_armCtrlFreq);
m_cmdTrqLpf.init(1, g_cmdJntTrqLpfCutoffFreq, g_armCtrlFreq);
m_curTrqLpf.init(1, g_curJntTrqLpfCutoffFreq, g_armCtrlFreq);

// driver init value
m_motorOutputs.m_controlWord:=DriverCtrlWord_INIT;
m_motorOutputs.m_opMode:=INT_TO_SINT(DriverOPMode_Pos);
m_motorOutputs.m_cmdCurrent:=0;
m_motorOutputs.m_cmdMotorEncoder:=m_motorInputs.m_motorEncoder;
END_METHOD

END_FUNCTION_BLOCK

// ---- FBs_Robots/FB_JointBase.TcPOU
FUNCTION_BLOCK FB_JointBase
VAR
	// motor IO
	m_motorInputs AT%I*	:ST_MotorInputs;
	m_motorOutputs AT%Q* :ST_MotorOutputs;
		
	// cycle time
	m_cycleTime :LREAL;
	
	// calibrated link encoder data
	m_minLinkEncoder :DINT;
	m_maxLinkEncoder :DINT;
	m_caliLinkEncoder :DINT;
	m_linkEncCaliJntPos :LREAL;
	m_linkEncZeroCross :INT;
	m_initMotorEnc : DINT;
	m_multiCycles :INT;
	
	// joint position from link encoder after power on
	m_initLinkPos :LREAL;
	
	// data for link encoder multiple cycles
	m_lastLinkEncoder :DINT;
	m_linkEncCycles:INT;
	
	// device paramters
	m_motorEncoderRes :DINT;
	m_linkEncoderRes :DINT;
	m_motorReduction :LREAL;
	m_linkEncoderReduction :LREAL;
	m_trqConst :LREAL;
	m_maxCurrent :LREAL;
	m_motorDir :INT;								
	m_linkEncoderDir :INT;
	m_minJntPos: LREAL;
	m_maxJntPos: LREAL;
	
	// macro defined data for quick calculation
	m_trq2CurrentRatio:LREAL;
	m_current2TrqRatio:LREAL;
	m_linkEnc2PosRatio :LREAL;
	m_motorEnc2PosRatio :LREAL;
	
	// joint data
	m_curMotorPos :LREAL;
	m_curLinkPos :LREAL;
	m_curJntPos	:LREAL;
	m_curJntVel :LREAL;
	m_curLinkVel :LREAL;
	m_curJntTrq :	LREAL;
	m_rawCurrent : LREAL;
	m_filtCurrent : LREAL;
	m_cmdJntPos :LREAL;
	m_cmdJntVel :LREAL;
	m_cmdJntTrq :LREAL;
	m_cmdCurrent : LREAL;
	m_lastJntPos :LREAL;
	m_lastLinkPos: LREAL;
	
	// velocity filter
	m_jntVelLpf :FB_LowPassFilter;
	m_linkVelLpf :FB_LowPassFilter;
	
	// current and command torque filter
	m_curTrqLpf : FB_LowPassFilter;
	m_cmdTrqLpf :FB_LowPassFilter;
	
END_VAR

PROPERTY cmdCurrent : LREAL
GET
cmdCurrent:=m_cmdCurrent;
END_GET
END_PROPERTY

METHOD PUBLIC disable : BOOL
VAR_INPUT
END_VAR
m_motorOutputs.m_controlWord:=DriverCtrlWord_INIT;
disable:=true;
END_METHOD

METHOD PUBLIC enable : BOOL
VAR_INPUT
END_VAR
IF DriverStatusWord_INIT = m_motorInputs.m_statusWord THEN
	m_motorOutputs.m_controlWord:=DriverCtrlWord_PREOP;
	enable := FALSE;
ELSIF DriverStatusWord_PREOP = m_motorInputs.m_statusWord THEN
	m_motorOutputs.m_controlWord:=DriverCtrlWord_OP;
	enable :=  FALSE;
ELSIF DriverStatusWord_OP = m_motorInputs.m_statusWord THEN
	enable :=  TRUE;
//ELSE
//	m_motorOutputs.m_controlWord:=DriverCtrlWord_INIT;
//	enable :=  FALSE;
END_IF
END_METHOD

PROPERTY filtCurrent : LREAL
GET
filtCurrent:=m_filtCurrent;
END_GET
END_PROPERTY

METHOD PUBLIC initJntPos : BOOL
VAR_INPUT
END_VAR
m_lastLinkEncoder :=m_motorInputs.m_linkEncoder;
m_linkEncCycles:=0;
m_curLinkPos :=linkEnc2Pos();
m_initLinkPos:=m_curLinkPos;
m_initMotorEnc :=m_motorInputs.m_motorEncoder;
m_curMotorPos:=motorEnc2Pos();
m_curJntPos := m_curMotorPos;
m_cmdJntPos :=m_curJntPos;	
m_lastJntPos :=m_curJntPos;
m_lastLinkPos := m_curLinkPos;

// filter init
m_jntVelLpf.init(1, g_curJntVelLpfCutoffFreq, g_armCtrlFreq);
m_linkVelLpf.init(1, g_curJntVelLpfCutoffFreq, g_armCtrlFreq);
END_METHOD

// reset the initial joint position with input value
METHOD PUBLIC initJntPosReset : BOOL
VAR_INPUT
	i_initLinkPos:LREAL;
END_VAR
m_initLinkPos:=i_initLinkPos;
m_initMotorEnc :=m_motorInputs.m_motorEncoder;
m_curMotorPos:=motorEnc2Pos();
m_curJntPos := m_curMotorPos;
m_cmdJntPos :=m_curJntPos;	
m_lastJntPos :=m_curJntPos;
m_lastLinkPos := m_curLinkPos;

// filter init
m_jntVelLpf.init(1, g_curJntVelLpfCutoffFreq, g_armCtrlFreq);
m_linkVelLpf.init(1, g_curJntVelLpfCutoffFreq, g_armCtrlFreq);
END_METHOD

PROPERTY initLinkPos : lreal
GET
initLinkPos:=m_initLinkPos;
END_GET
SET
m_initLinkPos:=initLinkPos;
END_SET
END_PROPERTY

METHOD PUBLIC isEnabled : BOOL
VAR_INPUT
END_VAR
isEnabled :=(DriverStatusWord_OP = m_motorInputs.m_statusWord);
END_METHOD

PROPERTY jntPos : LREAL
GET
jntPos := m_curJntPos;
END_GET
END_PROPERTY

PROPERTY jntTrq : LREAL
GET
jntTrq:=m_curJntTrq;
END_GET
END_PROPERTY

PROPERTY jntVel : LREAL
GET
jntVel := m_curJntVel;
END_GET
END_PROPERTY

METHOD PROTECTED linkEnc2Pos : LREAL
VAR_INPUT
END_VAR
VAR
	incLinkPos :LREAL;
	newLinkEnc :DINT;
END_VAR
// cycle check
IF 1=m_multiCycles THEN
	IF (m_motorInputs.m_linkEncoder - m_lastLinkEncoder)*m_linkEncoderDir < -m_linkEncoderRes/2 THEN
		m_linkEncCycles :=m_linkEncCycles+1;
	ELSIF (m_motorInputs.m_linkEncoder - m_lastLinkEncoder)*m_linkEncoderDir > m_linkEncoderRes/2 THEN
		m_linkEncCycles :=m_linkEncCycles-1;
	END_IF
END_IF
m_lastLinkEncoder:=m_motorInputs.m_linkEncoder;

// convert link encoder if joint cross zero
newLinkEnc := m_motorInputs.m_linkEncoder;
IF 1=m_linkEncZeroCross AND 0 = m_multiCycles THEN
	IF 1=m_linkEncoderDir AND m_motorInputs.m_linkEncoder < m_minLinkEncoder THEN
		newLinkEnc := m_motorInputs.m_linkEncoder + m_linkEncoderRes;
	ELSIF -1=m_linkEncoderDir AND m_motorInputs.m_linkEncoder < m_maxLinkEncoder THEN
		newLinkEnc := m_motorInputs.m_linkEncoder + m_linkEncoderRes;
	END_IF
END_IF

// motion from calibrated points
incLinkPos := (newLinkEnc-m_caliLinkEncoder)*m_linkEnc2PosRatio;

// absolute joint position
linkEnc2Pos := incLinkPos + m_linkEncCaliJntPos + 2*PI* m_linkEncCycles;
END_METHOD

PROPERTY PUBLIC linkPos : LREAL
GET
linkPos:=m_curLinkPos;
END_GET
END_PROPERTY

METHOD PROTECTED motorEnc2Pos : LREAL
VAR_INPUT
END_VAR
motorEnc2Pos:= (m_motorInputs.m_motorEncoder-m_initMotorEnc)* m_motorEnc2PosRatio +m_initLinkPos;
END_METHOD

PROPERTY PUBLIC motorPos : LREAL
GET
motorPos := m_curMotorPos;
END_GET
END_PROPERTY

METHOD PROTECTED motorPos2Enc : DINT
VAR_INPUT
	i_jntPos :LREAL;
END_VAR

VAR
END_VAR
motorPos2Enc := LREAL_TO_DINT((i_jntPos-m_initLinkPos)/m_motorEnc2PosRatio + m_initMotorEnc);
END_METHOD

PROPERTY rawCurrent : LREAL
GET
rawCurrent := m_rawCurrent;
END_GET
END_PROPERTY

METHOD PUBLIC updateCmds : BOOL
VAR_INPUT
	i_opMode : E_DriverOPMode;
	i_cmdPos :LREAL;
	i_cmdTrq :LREAL;
END_VAR
VAR
	filtCmdTrq :LREAL;
END_VAR
m_motorOutputs.m_opMode:=INT_TO_SINT( i_opMode);
// pos mode
IF i_opMode = DriverOPMode_Pos THEN
	m_motorOutputs.m_cmdCurrent:=0;
	m_cmdTrqLpf.reset();
//	i_cmdPos:=LIMIT(m_minJntPos, i_cmdPos, m_maxJntPos);
	m_motorOutputs.m_cmdMotorEncoder :=motorPos2Enc(i_cmdPos);
ELSIF i_opMode = DriverOPMode_Trq THEN
	filtCmdTrq:=m_cmdTrqLpf.run(i_cmdTrq);
	m_motorOutputs.m_cmdCurrent:=LREAL_TO_DINT(LIMIT(-m_maxCurrent, filtCmdTrq*m_trq2CurrentRatio,m_maxCurrent));
	m_motorOutputs.m_cmdMotorEncoder :=m_motorInputs.m_motorEncoder; 
END_IF
m_cmdCurrent:=m_motorOutputs.m_cmdCurrent;
END_METHOD

METHOD PUBLIC updateStatus : BOOL
VAR_INPUT
END_VAR
// compute joint position
m_curLinkPos:= linkEnc2Pos();
m_curMotorPos:=motorEnc2Pos();
m_curJntPos := m_curMotorPos;

// compute joint velocity
m_curJntVel:= (m_curJntPos-m_lastJntPos)/m_cycleTime;
m_curJntVel := m_jntVelLpf.run(m_curJntVel);
m_lastJntPos :=m_curJntPos;

// compute link velocity
m_curLinkVel := (m_curLinkPos-m_lastLinkPos)/m_cycleTime;
m_curLinkVel := m_linkVelLpf.run(m_curLinkVel);
m_lastLinkPos := m_curLinkPos;

// current and torque
m_rawCurrent := m_motorInputs.m_current;
m_filtCurrent := m_curTrqLpf.run(m_rawCurrent);
m_curJntTrq := m_filtCurrent * m_current2TrqRatio;
END_METHOD

END_FUNCTION_BLOCK

// ---- AgiMaths/atan2.TcPOU
FUNCTION atan2 : LREAL
VAR_INPUT
	y:LREAL;
	x:lreal;	
END_VAR
VAR
END_VAR


IF (x>0 AND y>0) THEN  //第1象限
	atan2:=ATAN(y/x);
ELSIF(x<0 AND y>0) THEN  //第2象限
	atan2:=ATAN(y/x)+pi;

ELSIF(x<0 AND y<0) THEN  //第3象限
	atan2:=ATAN(y/x)-pi;

ELSIF(x>0 AND y<0) THEN  //第4象限
	atan2:=ATAN(y/x);

ELSIF (x=0 AND y>0) THEN  //正Y轴
	atan2:=pi/2;

ELSIF (x=0 AND y<0) THEN  //负Y轴
	atan2:=-pi/2;
	
ELSIF (x>0 AND y=0) THEN  //正X轴
	atan2:=0;

ELSIF (x<0 AND y=0) THEN  //负X轴
	atan2:=pi;	
	
END_IF

END_FUNCTION

// ---- AgiMaths/MatrixLib/matMultiVec.TcPOU
// vecB = matA * vecA
FUNCTION matMultiVec : bool
VAR_IN_OUT CONSTANT
	matA :ARRAY[*,*] OF LREAL;//m*n
	vecA:ARRAY[*] OF LREAL; // n*1
END_VAR
VAR_IN_OUT 
		vecB :ARRAY[*] OF LREAL;
END_VAR
VAR
	m,n :DINT;
	i,j, k :DINT;
 
END_VAR

m:=UPPER_BOUND(matA,1);
n:= UPPER_BOUND(matA,2);
ASSERT(UPPER_BOUND(vecA,1)=n);
ASSERT(UPPER_BOUND(vecB,1)=m);
FOR i:=1 TO m DO
	vecB[i]:=0.0;
	FOR j:=1 TO n DO
		vecB[i]:=vecB[i]+matA[i,j]*vecA[j];
	END_FOR
END_FOR

END_FUNCTION

// ---- SafetyCheck/ASSERT.TcPOU
// this function is used to check if input statament is true.
// if false, the code will trigger a zero-devide exception and stop the whole program by PLC
FUNCTION ASSERT : BOOL
VAR_INPUT
	statement:BOOL;
END_VAR
VAR
	zero:INT :=0;
	res :REAL:=0;
END_VAR

IF NOT(statement) THEN
	res := 1/zero;
END_IF

ASSERT := true;

END_FUNCTION

// ---- FBs_Auxiliary/FB_MSCtrlTriggerCheck.TcPOU
//NOTE：this block would stop checking once a trigger is detected. 
//	re-init this block if want to start another check
FUNCTION_BLOCK FB_MSCtrlTriggerCheck
VAR_INPUT
END_VAR
VAR_OUTPUT
END_VAR
VAR
	// flag if master-slave control is enabled
	m_MSCtrlTrigger :BOOL;
	
	// block run time
	m_timePeriod :LREAL;
	
	// gripper state: 0-init, 1-open, 2-close, 3-reopen, 1-2-3 for one grip action
	m_gripperState :INT;
	
	// grip action counts
	m_gripActionCounts :INT;

	// two grip action within this duration indication to enable master-slave control
	m_checkDuration : LREAL;
	
	// time cycle
	m_timeCycle :LREAL;
	
	// time stamp for first grip
	m_firstGripTime :LREAL;
	
	// angle threshold indicating gripper open
	m_openAngThres :LREAL := g_maxGripAngle * 0.5;
	
	// angle threshold indicating gripper close
	m_closeAngThres :LREAL := 2.0 *g_deg2rad;
END_VAR

METHOD gripActionCheck : BOOL
VAR_INPUT
	i_gripAngle :LREAL;
END_VAR
gripActionCheck:=false;
CASE m_gripperState OF 
	0:
		IF i_gripAngle > m_openAngThres THEN
			m_gripperState :=1;
		END_IF
		
	1: IF i_gripAngle < m_openAngThres AND i_gripAngle > m_closeAngThres THEN
			m_gripperState:=2;
		END_IF
		
	2:
		IF i_gripAngle < m_closeAngThres THEN
			m_gripperState :=3;
		ELSIF i_gripAngle > m_openAngThres THEN
			m_gripperState :=1;
		END_IF
	3:
		IF i_gripAngle > m_openAngThres THEN
			m_gripperState :=4;
		END_IF
	4:
		gripActionCheck:=TRUE;
		m_gripperState:=0;
END_CASE
END_METHOD

METHOD init : BOOL
VAR_INPUT
	i_timeCycle :LREAL;
	i_checkDuration :LREAL;
END_VAR
m_timeCycle :=i_timeCycle;
m_checkDuration := i_checkDuration;
m_gripperState:=0;
m_gripActionCounts:=0;
m_MSCtrlTrigger :=false;
END_METHOD

METHOD reset : BOOL
VAR_INPUT
END_VAR
m_gripperState:=0;
m_gripActionCounts:=0;
m_MSCtrlTrigger :=FALSE;
END_METHOD

METHOD run : BOOL
VAR_INPUT
	i_gripAngle :LREAL;
END_VAR
IF m_MSCtrlTrigger THEN
	run := TRUE;
	RETURN;
END_IF

m_timePeriod := m_timePeriod + m_timeCycle;

// detect one grip action
IF gripActionCheck(i_gripAngle) THEN
	m_gripActionCounts:=m_gripActionCounts+1;
	
	// first grip
	IF 1=m_gripActionCounts THEN
		m_firstGripTime := m_timePeriod;
	ELSIF m_gripActionCounts>=2 THEN
		// second grip and trigger success
		IF m_timePeriod - m_firstGripTime < m_checkDuration THEN
			m_MSCtrlTrigger :=TRUE;
		ELSE
		// set second grip as new first one
			m_gripActionCounts:=1;
			m_firstGripTime:=m_timePeriod;
		END_IF
	END_IF
END_IF


run :=FALSE;
END_METHOD

END_FUNCTION_BLOCK

// ---- FBs_StateControllers/FB_StateCtrlError.TcPOU
// Brief: Master Arm Error Hold
FUNCTION_BLOCK PUBLIC FB_StateCtrlError EXTENDS FB_MasterArmCtrlBase
VAR_INPUT
END_VAR
VAR_OUTPUT
END_VAR
VAR
END_VAR

METHOD PUBLIC init : BOOL
VAR_IN_OUT CONSTANT
	i_masterArm	:FB_MasterArm;
END_VAR
VAR_IN_OUT 
	r_masterArmCtrlCmd :ST_ArmCtrlCmds;
END_VAR

VAR
	i:INT;
END_VAR
SUPER^.Init(i_masterArm,r_masterArmCtrlCmd);

//disable joints which is error
FOR i := 1 TO g_mJntNum DO
	IF SafetyCheck.m_SafetyCheck.m_jntErrFlag[i_masterArm.armIdx, i, 2] OR SafetyCheck.m_SafetyCheck.m_jntErrFlag[i_masterArm.armIdx, i, 3] THEN
		m_jntEnableFlag[i] := 0;
	ELSE
		m_jntEnableFlag[i] := 1;
	END_IF
END_FOR

// update commands to arm
copyCmds(r_masterArmCtrlCmd);
END_METHOD

END_FUNCTION_BLOCK

// ---- FBs_StateControllers/FB_MasterArmCtrlBase.TcPOU
// Master Arm Base Controller, Hold at Current Posture
FUNCTION_BLOCK FB_MasterArmCtrlBase IMPLEMENTS I_MasterArmCtrl
VAR_INPUT
END_VAR
VAR_OUTPUT
END_VAR
VAR
	// flag if the controller has finished all its jobs
	m_isFinished:BOOL:=FALSE;
	
	// controller execute time period
	m_timePeriod :LREAL:=0;
	
	// flag to hold last commands
	m_holdLastCmds :BOOL := FALSE;
	
	// arm control data
	m_cmdJntPos : VEC7d;
	m_cmdJntVel : VEC7d;
	m_cmdJntAcc : VEC7d;
	m_cmdJntTrq : VEC7d;
	m_jntOPMode : Vec7i;
	m_jntEnableFlag :Vec7i;
	m_cmdCartPose : ST_Frame;
	m_cmdCartTwist : Vec6d;
END_VAR

// override this function in each exact controller
METHOD PROTECTED calcCmdJntPos : BOOL

VAR_IN_OUT CONSTANT
	i_slaveIdx :INT;
	i_shoulderPose :ST_Frame;
	i_masterArm :FB_MasterArm;
	i_slaveStatus :ST_SlaveStatus;
END_VAR
END_METHOD

// override this function in each exact controller
METHOD PROTECTED calcCmdJntTrq : BOOL

VAR_IN_OUT CONSTANT
	i_slaveIdx :INT;
	i_shoulderPose :ST_Frame;
	i_masterArm :FB_MasterArm;
	i_slaveStatus :ST_SlaveStatus;
END_VAR
// set joint torque to zero in default
m_cmdJntTrq := g_zeroVec7d;
END_METHOD

METHOD checkToHoldLastCmds : BOOL
VAR_IN_OUT CONSTANT
	i_masterArm :FB_MasterArm;
END_VAR
VAR
	j:INT;
	maxJntErr:LREAL;
	jntCtrlErr:Vec7d;
END_VAR
// check if to hold the command joint position unchanged
vecSub(i_masterArm.m_cmdJntPos, i_masterArm.m_curJntPos,jntCtrlErr);
maxJntErr:=0.0;
FOR j:=1 TO g_mJntNum DO
	maxJntErr:= MAX(maxJntErr, ABS(jntCtrlErr[j]));
END_FOR

checkToHoldLastCmds := (maxJntErr<g_jntCtrlErrForCmdHold);
END_METHOD

METHOD copyCmds : BOOL
VAR_IN_OUT 
	r_masterArmCtrlCmd :ST_ArmCtrlCmds;
END_VAR
r_masterArmCtrlCmd.m_jntEnableFlag :=m_jntEnableFlag;
r_masterArmCtrlCmd.m_cmdCartPose:=m_cmdCartPose;
r_masterArmCtrlCmd.m_cmdCartTwist:=m_cmdCartTwist;
r_masterArmCtrlCmd.m_cmdJntPos:=m_cmdJntPos;
r_masterArmCtrlCmd.m_cmdJntVel:=m_cmdJntVel;
r_masterArmCtrlCmd.m_cmdJntAcc:=m_cmdJntAcc;
r_masterArmCtrlCmd.m_cmdJntTrq:=m_cmdJntTrq;
r_masterArmCtrlCmd.m_jntOPMode:=m_jntOPMode;
END_METHOD

// override this function in each exact controller
// NOTICE: set joint control mode here, and do some initialization if needed
METHOD PUBLIC init : BOOL
VAR_IN_OUT CONSTANT
	i_masterArm	:FB_MasterArm;
END_VAR
VAR_IN_OUT 
	r_masterArmCtrlCmd :ST_ArmCtrlCmds;
END_VAR
m_timePeriod:=0;
m_jntEnableFlag :=g_onesVec7i;
m_jntOPMode:=g_allPosMode;
m_cmdCartPose:=i_masterArm.curCartPose;
m_cmdCartTwist:=g_zeroVec6d;
IF FALSE = m_holdLastCmds THEN
	m_cmdJntPos:=i_masterArm.curJntPos;
ELSE 
	m_cmdJntPos := r_masterArmCtrlCmd.m_cmdJntPos;
END_IF
m_cmdJntVel:=g_zeroVec7d;
m_cmdJntAcc:=g_zeroVec7d;
m_cmdJntTrq:=g_zeroVec7d;

// update commands to arm
copyCmds(r_masterArmCtrlCmd);
END_METHOD

PROPERTY isFinished : BOOL
GET
isFinished:=m_isFinished;
END_GET
END_PROPERTY

{warning '添加方法实现'}
METHOD reset : BOOL
m_isFinished:=FALSE;
END_METHOD

{warning '添加方法实现'}
METHOD run : BOOL

VAR_IN_OUT CONSTANT
	i_slaveIdx :INT;
	i_shoulderPose :ST_Frame;
	i_masterArm :FB_MasterArm;
	i_slaveStatus :ST_SlaveStatus;
END_VAR
VAR_IN_OUT
	r_masterArmCtrlCmd :ST_ArmCtrlCmds;
END_VAR
VAR
	i:INT;
END_VAR
IF m_isFinished THEN
	RETURN;
END_IF

// check if arm enabled
IF FALSE = i_masterArm.isEnabled(m_jntEnableFlag) THEN
	RETURN;
END_IF

// calculate command joint position--Motion control
calcCmdJntPos(i_slaveIdx, i_shoulderPose, i_masterArm,i_slaveStatus);

// calculate command joint torque -- Force control
calcCmdJntTrq(i_slaveIdx, i_shoulderPose, i_masterArm,i_slaveStatus);

// update commands to arm
copyCmds(r_masterArmCtrlCmd);

// update time period
m_timePeriod := m_timePeriod+g_armCtrlCycleTime;
END_METHOD

PROPERTY timePeriod : Lreal
GET
timePeriod := m_timePeriod;
END_GET
END_PROPERTY

END_FUNCTION_BLOCK

// ---- AgiMaths/MatrixLib/vecSub.TcPOU
// C = A - B;
FUNCTION vecSub : BOOL
VAR_IN_OUT CONSTANT
	vecA :ARRAY[*] OF LREAL;
	vecB :ARRAY[*] OF LREAL;
END_VAR

VAR_IN_OUT 
	vecC :ARRAY[*] OF LREAL;
END_VAR

VAR
	m :DINT;
	i:DINT;
 
END_VAR

m:=UPPER_BOUND(VecA,1);
ASSERT(UPPER_BOUND(VecB,1)=m);
ASSERT(UPPER_BOUND(VecC,1)=m);

FOR i:=1 TO m DO
	vecC[i]:=vecA[i]-vecB[i];
END_FOR

END_FUNCTION

// ---- Mains/SafetyCheck.TcPOU
PROGRAM SafetyCheck
VAR
	i: INT;
	// master robot information, including arm status and cartesian data
	m_masterStatus AT %I* :ST_masterStatus;
	
	// master robot joint data
	m_masterJointData AT %I* :ST_masterJointData;
	
	//cart status
	m_cartStatus AT %I* :ST_CartStatus;
	
	//cart joint data
	m_cartJointData AT %I* :ST_cartJointData;
	
	// error check result
	m_safetyCheckData AT %Q* :ST_SafetyData;
	
	//stop botton
	m_stopButton AT %I*: BOOL;
	
	m_cartLockSignalLeft AT %I* :BOOL;
	m_cartLockSignalRight AT %I* :BOOL;
	
	m_initFlag:bool;
	
	m_SafetyCheck : Fb_SafetyCheck;
	m_checkVariable : ARRAY[1..g_maxNum] OF checkInputVariable;
	m_EtherCATCheck :ARRAY [1..g_maxNum,1..g_maxArmJoint] OF Fb_EtherCATCheck;
	m_errCode :ARRAY [1..3] OF UDINT;
	m_motorEncoderLast : ARRAY[1..g_maxNum,1..g_maxArmJoint] OF DINT;
	
	
	m_armsRS:ARRAY [1..g_maxArmNum,1..10] OF RS;//复位优先双稳态器
	m_cartRS:ARRAY [1..10] OF RS;//复位优先双稳态器
	
	// wait time before robot init  for ethercat to be statble 
	m_safetyCheckInitWaitTime : LREAL:=0;
	//error robot data record
	m_dataRecord : Fb_dataRecord;
END_VAR

// reset data
IF FALSE = m_initFlag  THEN
	FOR i:=1  TO g_mArmNum DO 
		m_safetyCheckData.m_masterErrFlag[i]:=FALSE;
	END_FOR
	FOR i:=1  TO 4 DO 
		m_safetyCheckData.m_cartErrFlag[i]:=FALSE;
	END_FOR
	m_initFlag:=TRUE;
END_IF


armSafetyCheckInputCast();

armSafetyCheckAllowed();

robotPromptMassageCast();

// wait communication to be stable
IF(m_safetyCheckInitWaitTime<g_robotSafetyCheckWaitTime) THEN
	m_safetyCheckInitWaitTime := m_safetyCheckInitWaitTime+g_cartCtrlCycleTime;
	RETURN;
END_IF

FOR i:=1  TO g_maxNum DO
	m_SafetyCheck.systemSafetyCheck(i,m_checkVariable,m_masterStatus,m_cartJointData,m_masterJointData);
END_FOR

//error flag to control
readErrFlag();

//Fault code for UI
m_SafetyCheck.errCodeUpdating();

//The fault code is sent to the UI
GVL_interactUI.g_errIdType3:=m_SafetyCheck.o_ErrCode[3];
GVL_interactUI.g_errIdType2:=m_SafetyCheck.o_ErrCode[2];
GVL_interactUI.g_errIdType1:=m_SafetyCheck.o_ErrCode[1];

//clear fault
IF GVL_interactUI.g_uiResetFault=1 THEN
	m_safetyCheck.errFlagReset();
	GVL_interactUI.g_uiResetFault :=0;
END_IF

//robot record information
m_dataRecord.run(m_checkVariable , m_cartStatus , m_cartJointData , m_masterStatus , m_masterJointData );

METHOD armSafetyCheckAllowed : BOOL
VAR_INPUT
END_VAR
VAR
	i , j : INT; 
END_VAR

FOR i := 1 TO g_maxArmNum DO
	FOR j := 1 TO g_maxArmJoint DO
		//fault code 16#3003 
		m_SafetyCheck.checkPermit[i].m_linkEncErr[j] := m_checkVariable[i].m_masterDriverInput[j].m_statusWord<>0;
		//fault code 16#3002 
		m_SafetyCheck.checkPermit[i].m_currentIsNotUpdate[j] :=m_checkVariable[i].m_masterDriverInput[j].m_statusWord<>0 ;
		//fault code 16#2002
		m_SafetyCheck.checkPermit[i].m_armJntFollowErr[j] := m_masterStatus.m_armState[j] = MasterArmState_Home OR m_masterStatus.m_armState[j] = MasterArmState_MasterSlave;//m_checkVariable[i].m_masterDriverInput[j].m_statusWord = DriverStatusWord_OP ;
		//fault code 16#3002
		m_SafetyCheck.checkPermit[i].m_jntStatusErr[j] := TRUE;
		//fault code 16#3004
		m_SafetyCheck.checkPermit[i].m_driveErr[j] := TRUE;
		//fault code 16#3005
		m_SafetyCheck.checkPermit[i].m_armJntEncErr[j] := TRUE;
		//fault code 16#2003
		m_SafetyCheck.checkPermit[i].m_jntVelErr[j] := TRUE;
		//fault code 16#2004
		//m_SafetyCheck.checkPermit[i].m_spacePoseErr[j] := m_masterStatus.m_armState[i] = SlaveArmState_MasterSlave AND  norm(m_masterStatus.m_masterSlavePoseError[i])<g_smallNum;
		//fault code 16#2005
		m_SafetyCheck.checkPermit[i].m_jntCurrentErr[j] := TRUE;
	END_FOR
END_FOR
END_METHOD

METHOD armSafetyCheckInputCast : BOOL
VAR_INPUT
END_VAR

VAR
	i , j: INT; 
END_VAR

FOR i := 1 TO g_maxArmNum DO
	//stop button and ui stop 
	m_checkVariable[i].PCStopButton := GVL_interactUI.g_masterStopButton;
	m_checkVariable[i].SlaveStopButton := MasterArmControl.m_masterInputDataPool.m_slaveStatus.m_slaveStopButton;
	m_checkVariable[i].MasterStopButton := m_stopButton;
	m_checkVariable[i].m_spacePoseErr := m_SafetyCheck.poseErrCheck(m_masterStatus.m_cmdArmPose[i], m_masterStatus.m_curArmPose[i] );
	FOR j:=1 TO  g_mJntNum DO 		
		m_checkVariable[i].m_masterDriverInput[j] := MasterArmControl.m_masterRobot.m_masterArms[i].m_joints[j].m_motorInputs;
		m_checkVariable[i].m_masterDriverOutput[j] := MasterArmControl.m_masterRobot.m_masterArms[i].m_joints[j].m_motorOutputs;
		m_checkVariable[i].m_EtherCATState[j] := m_EtherCATCheck[i,j].EtherCATVerify(g_ArmNetID[i],g_JointNetPort[i,j]);
		m_checkVariable[i].m_motorEncSaltaValue[j] := ABS(MasterArmControl.m_masterRobot.m_masterArms[i].m_joints[j].m_motorInputs.m_motorEncoder - m_motorEncoderLast[i,j]);
		m_motorEncoderLast[i,j] := MasterArmControl.m_masterRobot.m_masterArms[i].m_joints[j].m_motorInputs.m_motorEncoder;
		//The sum of the square of the motor current
		g_motorCurrentLimit[j] := EXPT((GVL_ArmJointParameters.g_motorMaxCurrent[j]/1000),2)*15000;
		IF ABS(m_checkVariable[i].m_masterDriverInput[j].m_current) > GVL_ArmJointParameters.g_motorMaxCurrent[j] THEN
			m_checkVariable[i].m_motorCurrentIntegral[j] := m_checkVariable[i].m_motorCurrentIntegral[j] + ABS (EXPT((DINT_TO_LREAL(m_checkVariable[i].m_masterDriverInput[j].m_current)/1000),2));
		ELSE
			m_checkVariable[i].m_motorCurrentIntegral[j] := 0;
		END_IF
	END_FOR
END_FOR

FOR j:=1 TO  g_maxCartJoint DO
	m_checkVariable[g_cartNum].PCStopButton := GVL_interactUI.g_masterStopButton;
	m_checkVariable[g_cartNum].MasterStopButton := m_stopButton;
	m_checkVariable[g_cartNum].m_cartDriverInput[j] := CartControl.m_masterCart.m_cartJoints[j].m_motorInputs;
	m_checkVariable[g_cartNum].m_cartDriverOutput[j] := CartControl.m_masterCart.m_cartJoints[j].m_motorOutputs;
	m_checkVariable[g_cartNum].m_cartEtherCATState[j] := m_EtherCATCheck[g_cartNum,j].EtherCATVerify(g_cartNetID,g_cartJointNetPort[j]);
END_FOR
END_METHOD

METHOD readErrFlag : BOOL
VAR_INPUT
END_VAR

FOR i:=1  TO g_mArmNum DO
	m_safetyCheckData.m_masterErrFlag[i] := m_SafetyCheck.m_armErrFlag[i,2] OR m_SafetyCheck.m_armErrFlag[i,3];
END_FOR
FOR i:=1  TO g_maxCartJoint DO
	m_safetyCheckData.m_cartErrFlag[i] := m_SafetyCheck.m_jntErrFlag[g_cartNum,i,2] OR m_SafetyCheck.m_jntErrFlag[g_cartNum,i,3] OR m_SafetyCheck.m_jntErrFlag[g_cartNum,0,2] OR m_SafetyCheck.m_jntErrFlag[g_cartNum,0,3];
END_FOR
END_METHOD

METHOD robotPromptMassageCast : BOOL
VAR_IN_OUT CONSTANT
END_VAR

VAR
	i : INT;
	m_uiCtrlAdjustFlag : BOOL;
	m_uiCtrlJoystickEnable : BOOL;
	m_joysticksTrigger : BOOL;
END_VAR

FOR i := 1 TO g_mArmNum DO					
	//0*1012		
	m_armsRS[i,2](SET:=m_masterStatus.m_armState[i] = MasterArmState_Disable AND m_cartStatus.m_surgonReady, 
							RESET1:= NOT m_armsRS[i,2].SET, 
							Q1=> m_checkVariable[i].m_promptStatus[2]);
	m_checkVariable[i].m_promptLocation[2] := i;
						
	//0*1013				
	m_armsRS[i,3](SET:=m_masterStatus.m_armState[i] = MasterArmState_Matching AND NOT m_masterStatus.m_IKSuccess[i] AND m_masterStatus.m_timePeriod[i]>0.01, 
							RESET1:= NOT m_armsRS[i,3].SET, 
							Q1=> m_checkVariable[i].m_promptStatus[3]);
	m_checkVariable[i].m_promptLocation[3] := i;
	
	//0*1014	
	m_armsRS[i,4](SET:=m_masterStatus.m_armState[i] = MasterArmState_Matching AND m_masterStatus.m_IKSuccess[i] AND m_masterStatus.m_timePeriod[i]>10, 
							RESET1:= NOT m_armsRS[i,4].SET, 
							Q1=> m_checkVariable[i].m_promptStatus[4]);
	m_checkVariable[i].m_promptLocation[4] := i;

END_FOR

//0*1011
m_cartRS[1](SET:= m_masterStatus.m_matchedMasterArmIdx.left1ArmIdx <> GVL_interactUI.g_armDistributionInfo.m_leftMappingSlaveArm[1] OR m_masterStatus.m_matchedMasterArmIdx.left2ArmIdx <> GVL_interactUI.g_armDistributionInfo.m_leftMappingSlaveArm[2], 
						RESET1:= NOT m_cartRS[1].SET, 
						Q1=> m_checkVariable[g_cartNum].m_promptStatus[1]);
m_checkVariable[g_cartNum].m_promptLocation[1] := 16#0B;

//0*1015
m_cartRS[5](SET:=NOT m_masterStatus.m_slaveOnLine, 
						RESET1:= NOT m_cartRS[5].SET, 
						Q1=> m_checkVariable[g_cartNum].m_promptStatus[5]);
m_checkVariable[g_cartNum].m_promptLocation[5] := g_cartNum;

//0*1016
m_cartRS[6](SET:=m_cartStatus.m_consoleInAdjust AND m_cartStatus.m_surgonReady, 
						RESET1:= NOT m_cartRS[6].SET, 
						Q1=> m_checkVariable[g_cartNum].m_promptStatus[6]);
m_checkVariable[g_cartNum].m_promptLocation[6] := g_cartNum;

//0*1017
m_cartRS[7](SET:=NOT (m_cartLockSignalLeft OR m_cartLockSignalRight ), 
						RESET1:= NOT m_cartRS[7].SET, 
						Q1=> m_checkVariable[g_cartNum].m_promptStatus[7]);
m_checkVariable[g_cartNum].m_promptLocation[7] := g_cartNum;
END_METHOD

END_PROGRAM

// ---- SafetyCheck/Fb_SafetyCheck.TcPOU
FUNCTION_BLOCK Fb_SafetyCheck
VAR_INPUT
END_VAR
VAR_OUTPUT
END_VAR
VAR
	i, j:INT;
	m_checkDelay :ARRAY[1..g_maxNum] OF checkDelay;
	m_checkDelayTime :checkDelayTime;
	m_checkPermit:ARRAY[1..g_maxNum] OF  checkPermit;
	
	m_jntErrFlag:ARRAY[1..g_maxNum,0..g_maxArmJoint,1..3] OF BOOL;
	m_armErrFlag:ARRAY [1..g_maxNum,1..3] OF BOOL;
	m_errCode:UDINT;
	
	
	m_errNumType: ARRAY [1..3] OF INT;
	m_ArrayErrCodeType:ARRAY [1..3] OF ARRAY [0..100] OF UDINT;
	
	//The fault is sent to the UI at the frequency of 0.1S
	m_errCodeUpdateFlag: ARRAY [1..3] OF BOOL;
	m_errCodeUpdateTon: ARRAY [1..3] OF TON;
	
	m_curJntTorqueIOlast :ARRAY [1..g_maxArmNum] OF vec7di;  
	m_cmdJntPosLast : ARRAY [1..g_maxArmNum] OF vec7d;  
	m_cartCurJntTorqueIOlast :ARRAY [1..4] OF LREAL;  
	m_cartCmdJntPosLast : ARRAY [1..4] OF LREAL; 
	o_ErrCode:ARRAY [1..3] OF UDINT;
		
	//error robot data record
	m_dataRecord : Fb_dataRecord;
	
	m_PromptMassBusy:BOOL;
	m_PromptFlag:ARRAY[1..g_maxNum,1..20] OF UINT;
	m_deleteCode:UDINT;
	
END_VAR


VAR CONSTANT
	m_codeUpdateDelay:TIME:=T#0.1S;
	
	//Fault level: 1 indicates  prompt message, 2 indicates a recoverable fault and 3 indicates an unrecoverable fault
	m_promptMessageLevel : UINT :=1;
	m_rcvLevel : UINT :=2;
	m_unrcvLevel : UINT :=3;
END_VAR

METHOD armSafetyCheck : BOOL
VAR_INPUT
	i_armId:UDINT;
	i_safetyCheckVar :ARRAY[1..g_maxNum] OF checkInputVariable;
	i_masterStatus :ST_MasterStatus;
	i_masterJointData : ST_MasterJointData;
END_VAR

VAR
	k:INT;
END_VAR

//驱动器状态监测、驱动器未连接
FOR i:=1 TO g_mJntNum BY 1 DO
	m_checkDelay[i_ArmId].T_jntStatusErr[i](IN:= (i_safetyCheckVar[i_ArmId].m_masterDriverInput[i].m_statusWord=0 AND m_checkPermit[i_ArmId].m_jntStatusErr[i]), PT:=m_checkDelayTime.Ti_jntStatusErr , Q=> , ET=> );
	IF m_checkDelay[i_ArmId].T_jntStatusErr[i].Q  THEN
		errCodeAssign(i_ArmId, i_ArmId,  0, i, 16#3002 ,m_unrcvLevel );
	END_IF
END_FOR



//关节编码器监测
FOR i:=1 TO g_mJntNum BY 1 DO
	m_checkDelay[i_ArmId].T_linkEncErr[i](IN:= (i_safetyCheckVar[i_ArmId].m_masterDriverInput[i].m_linkEncoder=g_maxLinkEnc OR i_safetyCheckVar[i_ArmId].m_masterDriverInput[i].m_linkEncoder=g_minLinkEnc) AND m_checkPermit[i_ArmId].m_linkEncErr[i], PT:=m_checkDelayTime.Ti_linkEncErr , Q=> , ET=> );
	IF m_checkDelay[i_ArmId].T_linkEncErr[i].Q THEN
		errCodeAssign(i_ArmId, i_ArmId,  0, i,  16#3003 ,m_unrcvLevel );
	END_IF
END_FOR


//驱动器错误检测
FOR i:=1 TO g_mJntNum BY 1 DO
	m_checkDelay[i_ArmId].T_DriveErr[i](IN:= (i_safetyCheckVar[i_ArmId].m_masterDriverInput[i].m_driverError AND 16#20)=g_driveErrWord AND m_checkPermit[i_ArmId].m_driveErr[i] , PT:=m_checkDelayTime.Ti_driveErr , Q=> , ET=> );
	IF m_checkDelay[i_ArmId].T_DriveErr[i].Q THEN
		errCodeAssign(i_ArmId, i_ArmId,  0, i, 16#3004 ,m_unrcvLevel );
	END_IF
END_FOR


//双编码器偏差过大检测
FOR i:=1 TO g_mJntNum BY 1 DO
	m_checkDelay[i_ArmId].T_armJntEncErr[i](IN:= ABS(i_masterJointData.m_curLinkPos[i_armId][i]-i_masterJointData.m_curJntPos[i_armId][i])>=g_armMaxJntEncErr[i] AND m_checkPermit[i_ArmId].m_armJntEncErr[i], PT:=m_checkDelayTime.Ti_armJntEncErr , Q=> , ET=> );
	IF m_checkDelay[i_ArmId].T_armJntEncErr[i].Q THEN
		errCodeAssign( i_ArmId, i_ArmId,  0, i, 16#3005, m_unrcvLevel );
	END_IF
END_FOR


//关节运动超限位
FOR i:=1 TO g_mJntNum BY 1 DO
	m_checkDelay[i_armId].T_outOfLimit[i](IN:= i_masterJointData.m_curJntPos[i_armId][i]>= (g_maxJntPos[i_armId,i] + g_armJntPosLimitBuffer[i]) OR i_masterJointData.m_curJntPos[i_armId][i]<=(g_minJntPos[i_armId,i] - g_armJntPosLimitBuffer[i]) AND m_checkPermit[i_ArmId].m_outOfLimit[i], PT:=m_checkDelayTime.Ti_outofLimit , Q=> , ET=> );
	IF m_checkDelay[i_armId].T_outOfLimit[i].Q THEN
		errCodeAssign(i_armId, i_ArmId,  0, i, 16#3006, m_unrcvLevel );
	END_IF
END_FOR


//驱动器内部通讯错误
FOR i:=1 TO g_mJntNum BY 1 DO
	m_checkDelay[i_armId].T_currentIsNotUpdate[i](IN:= (i_safetyCheckVar[i_ArmId].m_masterDriverInput[i].m_current=m_curJntTorqueIOlast[i_ArmId][i] AND m_checkPermit[i_ArmId].m_currentIsNotUpdate[i]), PT:=m_checkDelayTime.Ti_currentIsNotUpdate , Q=> , ET=> );
	IF  m_checkDelay[i_armId].T_currentIsNotUpdate[i].Q THEN
		errCodeAssign(i_armId, i_ArmId,  0, i, 16#3009 ,m_unrcvLevel );
	END_IF
	m_curJntTorqueIOlast[i_armId][i]:=i_safetyCheckVar[i_armId].m_masterDriverInput[i].m_current;
END_FOR


//关节跟随误差过大
FOR i:=1 TO g_mJntNum BY 1 DO
	m_checkDelay[i_ArmId].T_armJntFollowErr[i](IN:= ABS(i_masterJointData.m_cmdJntPos[i_armId][i]- i_masterJointData.m_curJntPos[i_armId][i])>g_armMaxJntFollowErr[i]  AND m_checkPermit[i_ArmId].m_armJntFollowErr[i], PT:=m_checkDelayTime.Ti_armJntFollowErr , Q=> , ET=> );
	IF m_checkDelay[i_ArmId].T_armJntFollowErr[i].Q THEN
		errCodeAssign(i_ArmId, i_ArmId,  0, i, 16#2002, m_rcvLevel );
	END_IF
END_FOR


//笛卡尔空间指令与位置偏差检测
//FOR i:=1 TO 6 BY 1 DO
//	m_checkDelay[i_ArmId].T_spacePoseErr[i](IN:= i_safetyCheckVar[i_ArmId].m_spacePoseErr[i]> g_maxCartPoseErr[i] AND m_checkPermit[i_ArmId].m_spacePoseErr[i], PT:=m_checkDelayTime.Ti_spacePoseErr , Q=> , ET=> );
//	IF m_checkDelay[i_ArmId].T_spacePoseErr[i].Q THEN
//		errCodeAssign(i_ArmId, i_ArmId, 1, i, 16#2004, m_rcvLevel );
//	END_IF
//END_FOR


//current overrun check
FOR i:=1 TO g_mJntNum BY 1 DO
	m_checkDelay[i_armId].T_jntCurrentErr[i](IN:= ABS(i_safetyCheckVar[i_armId].m_motorCurrentIntegral[i])>g_motorCurrentLimit[i] AND m_checkPermit[i_ArmId].m_jntCurrentErr[i], PT:=m_checkDelayTime.Ti_jntCurrentErr , Q=> , ET=> );
	IF m_checkDelay[i_armId].T_jntCurrentErr[i].Q THEN
		errCodeAssign(i_armId, i_ArmId,  0, i, 16#2005, m_rcvLevel );
	END_IF
END_FOR


//Ethercat communication check
FOR i:=1 TO g_mJntNum BY 1 DO
	IF NOT i_safetyCheckVar[i_ArmId].m_EtherCATState[i].EtherCATState THEN
		errCodeAssign(i_ArmId, i_ArmId, 0, i, 16#2006, m_rcvLevel );
	END_IF
END_FOR


//self check failure
IF i_masterStatus.m_armState[i_armId] = MasterArmState_Home AND i_masterStatus.m_timePeriod[i] > g_selfCheckTimeLimit THEN//i_safetyCheckVar[i_armId].m_selfCheckFail THEN
	errCodeAssign(i_armId, i_ArmId,  0, i, 16#2008, m_rcvLevel );
END_IF

//motor encoder mutation detection
FOR i:=1 TO g_mJntNum BY 1 DO
	IF i_safetyCheckVar[i_armId].m_motorEncSaltaValue[i]>g_maxJntCurSalta[i] THEN
		errCodeAssign(i_armId, i_ArmId+3, 0, i, 16#200C, m_rcvLevel );
	END_IF
END_FOR

//master hall anomaly
IF i_masterStatus.m_gripHallSensor[i_armId] = 0 THEN
	errCodeAssign(i_armId, i_ArmId+3, 0, i, 16#200E, m_rcvLevel );
END_IF
END_METHOD

METHOD arrayDeleteFrist : ARRAY [0..100] OF UDINT;
VAR_INPUT
	i_array:ARRAY [0..100] OF UDINT;
END_VAR

VAR
	k:INT;
END_VAR

arrayDeleteFrist[100]:=0;

FOR k:=0 TO 99 BY 1 DO
	arrayDeleteFrist[k]:=i_array[k+1];
END_FOR
END_METHOD

METHOD arrayDeleteInput : BOOL
VAR_INPUT
	i_Array:ARRAY[0..100] OF UDINT;
	i_DeleteCode:UDINT;
END_VAR

VAR_OUTPUT
	o_Array:ARRAY[0..100] OF UDINT;
	
END_VAR

VAR
	i:INT;
	Falg:BOOL;
END_VAR

FOR i:=0 TO 20 BY 1 DO 
	IF i_Array[i]=i_DeleteCode THEN
		Falg:=TRUE;
	END_IF
	
	IF Falg=TRUE THEN
		o_Array[i]:=i_Array[i+1];
	ELSE
		o_Array[i]:=i_Array[i];
	END_IF
END_FOR
o_Array[20]:=0;
END_METHOD

METHOD arrayFIFO : ARRAY [0..100] OF  UDINT
VAR_INPUT
	i_array:ARRAY[0..100] OF UDINT;
	i_newData:UDINT;
END_VAR

VAR
	i:INT;
END_VAR

FOR i:=0 TO 20 BY 1 DO
	arrayFIFO[i+1]:=i_array[i];
END_FOR

arrayFIFO[0]:=i_newData;
END_METHOD

METHOD arrayFILO : ARRAY [0..100] OF  UDINT
VAR_INPUT
	i_array:ARRAY[0..100] OF UDINT;
	i_newData:UDINT;
END_VAR

VAR
	i:INT;
END_VAR

FOR i:=0 TO 20 BY 1 DO
	arrayFILO[i]:=i_array[i];
	IF i_array[i]=0 THEN
		arrayFILO[i]:=i_newData;
		EXIT;
	END_IF
END_FOR
END_METHOD

METHOD cartSafetyCheck : BOOL
VAR_INPUT
	i_armId:UDINT;
	i_safetyCheckVar : checkInputVariable;
	i_cartJointData : ST_CartJointData;
END_VAR


VAR
	k:INT;
END_VAR


//驱动器状态监测、驱动器未连接
FOR i:=1 TO g_maxCartJoint BY 1 DO
	m_checkDelay[i_armId].T_cartJntStatusErr[i](IN:= (i_safetyCheckVar.m_cartDriverInput[i].m_statusWord=0 AND m_checkPermit[i_ArmId].m_cartJntStatus[i]), PT:=m_checkDelayTime.Ti_CarJntStatus , Q=> , ET=> );
	IF m_checkDelay[i_armId].T_cartJntStatusErr[i].Q THEN
		errCodeAssign(i_armId, i_ArmId,  0, i, 16#3002 ,m_unrcvLevel );
	END_IF
END_FOR



//关节编码器监测
FOR i:=1 TO g_maxCartJoint BY 1 DO
	m_checkDelay[i_armId].T_cartLinkEncErr[i](IN:= (i_safetyCheckVar.m_cartDriverInput[i].m_linkEncoder=g_cartMaxLinkEnc[i] OR i_safetyCheckVar.m_cartDriverInput[i].m_linkEncoder=g_cartMinLinkEnc[i]) AND m_checkPermit[i_ArmId].m_cartJntEncErr[i], PT:=m_checkDelayTime.Ti_CarActSec , Q=> , ET=> );
	IF m_checkDelay[i_armId].T_cartLinkEncErr[i].Q THEN
		errCodeAssign(i_armId, i_ArmId,  0, i, 16#3003 ,m_unrcvLevel );
	END_IF
END_FOR


//驱动器错误检测
FOR i:=1 TO g_maxCartJoint BY 1 DO
	m_checkDelay[i_armId].T_cartDriveErr[i](IN:= (i_safetyCheckVar.m_cartDriverInput[i].m_driverError AND 16#20)=32 AND m_checkPermit[i_ArmId].m_cartDriveErr[i] , PT:=m_checkDelayTime.Ti_CarDriveErr , Q=> , ET=> );
	IF m_checkDelay[i_armId].T_cartDriveErr[i].Q THEN
		errCodeAssign(i_armId, i_ArmId,  0, i, 16#3004 ,m_unrcvLevel );
	END_IF
END_FOR



//台车双编码器偏差过大
FOR i:=1 TO g_maxCartJoint BY 1 DO
	m_checkDelay[i_armId].T_cartJntEncErr[i](IN:= ABS (i_cartJointData.m_curLinkPos[i]-i_cartJointData.m_curJntPos[i])>g_cartMaxJntEncErr[i] AND m_checkPermit[i_ArmId].m_cartJntEncErr[i], PT:=m_checkDelayTime.Ti_CarDualEncDev , Q=> , ET=> );
	IF m_checkDelay[i_armId].T_cartJntEncErr[i].Q THEN
		errCodeAssign(i_armId, i_ArmId,  0, i, 16#3005 ,m_unrcvLevel );
	END_IF
END_FOR


//关节运动超限位
FOR i:=1 TO g_maxCartJoint BY 1 DO
	m_checkDelay[i_armId].T_cartOutOfLimit[i](IN:= (i_cartJointData.m_curJntPos[i]>=g_cartMaxJntLimit[i] OR i_cartJointData.m_curJntPos[i]<=g_cartMinJntLimit[i]) AND m_checkPermit[i_ArmId].m_cartOutOfLimit[i] , PT:=m_checkDelayTime.Ti_CaroutofLimit , Q=> , ET=> );
	IF m_checkDelay[i_armId].T_cartOutOfLimit[i].Q THEN
		errCodeAssign(i_armId, i_ArmId,  0, i, 16#3006 ,m_unrcvLevel );
	END_IF
END_FOR


//驱动器内部通讯错误
FOR i:=1 TO g_maxCartJoint BY 1 DO
	m_checkDelay[i_armId].T_cartCurrentIsNotUpdate[i](IN:= (i_safetyCheckVar.m_cartDriverInput[i].m_current=m_cartCurJntTorqueIOlast[i] AND m_checkPermit[i_ArmId].m_cartCurrentIsNotUpdate[i]), PT:=m_checkDelayTime.Ti_CarTorMotor , Q=> , ET=> );
	IF m_checkDelay[i_armId].T_cartCurrentIsNotUpdate[i].Q THEN
		errCodeAssign(i_armId, i_ArmId,  0, i, 16#3009 ,m_unrcvLevel );
	END_IF
	m_cartCurJntTorqueIOlast[i]:=i_safetyCheckVar.m_cartDriverInput[i].m_current;
END_FOR


//关节跟随误差过大
FOR i:=1 TO g_maxCartJoint BY 1 DO
	m_checkDelay[i_armId].T_cartJntFollowErr[i](IN:= ABS(i_cartJointData.m_cmdJntPos[i]- i_cartJointData.m_curJntPos[i])>g_cartMaxJntFollowErr[i]  AND m_checkPermit[i_ArmId].m_cartFollowErr[i], PT:=m_checkDelayTime.Ti_CarFollowDev , Q=> , ET=> );
	IF m_checkDelay[i_armId].T_cartJntFollowErr[i].Q THEN
		errCodeAssign(i_armId, i_ArmId,  0, i, 16#2002 ,m_rcvLevel );
	END_IF
END_FOR


//关节速度监控
FOR i:=1 TO g_maxCartJoint BY 1 DO
	m_checkDelay[i_armId].T_cartJntVelErr[i](IN:= ABS(i_cartJointData.m_curJntVel[i])>g_cartMaxJntVel[i] AND m_checkPermit[i_ArmId].m_cartJntVelErr[i], PT:=m_checkDelayTime.Ti_CarJntVel , Q=> , ET=> );
	IF m_checkDelay[i_armId].T_cartJntVelErr[i].Q THEN
		errCodeAssign(i_armId, i_ArmId,  0, i, 16#2003 ,m_rcvLevel );
	END_IF
END_FOR


